# B&R Automation Studio project TD52 (part 91)

### Module_EngineGeneral.var - Module global variables
```iecst
VAR
	bAMM_2383 : BOOL := FALSE; (*ERROR: SAFETY - Exhaust gas backpressure high*) (*SAFETY PLC*) (*V04.14.00.00*)
	bAMM_2384 : BOOL := FALSE; (*ERROR: SAFETY - Speed deviation to ignition speed*) (*SAFETY PLC*) (*V04.14.00.00*)
	bAMM_2385 : BOOL := FALSE; (*ERROR: SAFETY - Ignition system failure*) (*SAFETY PLC*) (*V04.14.00.00*)
	bAMM_2386 : BOOL := FALSE; (*ERROR: SAFETY - Oil pressure minimum*) (*SAFETY PLC*) (*V04.14.00.00*)
	bAMM_2387 : BOOL := FALSE; (*ERROR: SAFETY - Oil pressure measuring signal failure*) (*SAFETY PLC*) (*V04.14.00.00*)
	bAMM_2388 : BOOL := FALSE; (*ERROR: SAFETY - Oil pressure implausible value*) (*SAFETY PLC*) (*V04.14.00.00*)
	bAMM_2389 : BOOL := FALSE; (*ERROR: SAFETY - Oil pressure deviation between the sensors*) (*SAFETY PLC*) (*V04.14.00.00*)
	bAMM_2390 : BOOL := FALSE; (*ERROR: SAFETY - Oil pressure maximum (sensor drift)*) (*SAFETY PLC*) (*V04.14.00.00*)
	bAMM_2391 : BOOL := FALSE; (*ERROR: SAFETY - Oil pressure sensor value frozen*) (*SAFETY PLC*) (*V04.14.00.00*)
	bAMM_2392 : BOOL := FALSE; (*ERROR: SAFETY - Oil pressure after pump maximum*) (*SAFETY PLC*) (*V04.14.00.00*)
	bAMM_2393 : BOOL := FALSE; (*ERROR: SAFETY - Oil pressure after pump measuring signal failure*) (*SAFETY PLC*) (*V04.14.00.00*)
	bAMM_2394 : BOOL := FALSE; (*ERROR: SAFETY - Oil pressure after pump implausible value*) (*SAFETY PLC*) (*V04.14.00.00*)
	bAMM_2395 : BOOL := FALSE; (*ERROR: SAFETY - Oil pressure after pump sensor value frozen*) (*SAFETY PLC*) (*V04.14.00.00*)
	bAMM_2396 : BOOL := FALSE; (*ERROR: SAFETY - Engine cooling water pressure minimum*) (*SAFETY PLC*) (*V04.14.00.00*)
	bAMM_2397 : BOOL := FALSE; (*ERROR: SAFETY - Engine cooling water pressure measuring signal failure*) (*SAFETY PLC*) (*V04.14.00.00*)
	bAMM_2398 : BOOL := FALSE; (*ERROR: SAFETY - Engine cooling water pressure deviation between the sensors*) (*SAFETY PLC*) (*V04.14.00.00*)
	bAMM_9408 : BOOL := FALSE; (*ERROR: SAFETY - Engine cooling water pressure maximum (sensor drift)*) (*SAFETY PLC*) (*V04.14.00.00*)
	bAMM_9409 : BOOL := FALSE; (*ERROR: SAFETY - Engine cooling water pressure sensor value frozen*) (*SAFETY PLC*) (*V04.14.00.00*)
	bAMM_9410 : BOOL := FALSE; (*ERROR: SAFETY - Engine cooling water pressure after pump maximum*) (*SAFETY PLC*) (*V04.14.00.00*)
	bAMM_9411 : BOOL := FALSE; (*ERROR: SAFETY - Engine cooling water pressure after pump measuring signal failure*) (*SAFETY PLC*) (*V04.14.00.00*)
	bAMM_9412 : BOOL := FALSE; (*ERROR: SAFETY - Engine cooling water pressure after pump sensor value frozen*) (*SAFETY PLC*) (*V04.14.00.00*)
	bAMM_9413 : BOOL := FALSE; (*ERROR: SAFETY - Generator circuit breaker opening failure*) (*SAFETY PLC*) (*V04.14.00.00*)
	bAMM_9414 : BOOL := FALSE; (*ERROR: SAFETY - Generator circuit breaker position feedback error*) (*SAFETY PLC*) (*V04.14.00.00*)
	bAMM_9415 : BOOL := FALSE; (*ERROR: SAFETY - Generator overload/short circuit*) (*SAFETY PLC*) (*V04.14.00.00*)
	bAMM_9416 : BOOL := FALSE; (*ERROR: SAFETY - Generator protection trip*) (*SAFETY PLC*) (*V04.14.00.00*)
	bAMM_9417 : BOOL := FALSE; (*ERROR: SAFETY - Collective fault in room ventilation*) (*SAFETY PLC*) (*V04.25.00.00*)
	bAMM_9418 : BOOL := FALSE; (*ERROR: SAFETY - Emergency stop push button - Module interface panel*) (*SAFETY PLC*) (*V04.14.00.00*)
	bAMM_9419 : BOOL := FALSE; (*ERROR: SAFETY - Emergency stop push button*) (*SAFETY PLC*) (*V04.14.00.00*)
	bAMM_9420 : BOOL := FALSE; (*ERROR: SAFETY - Safety loop 1 tripped - Module control panel*) (*SAFETY PLC*) (*V04.14.00.00*)
	bAMM_9421 : BOOL := FALSE; (*ERROR: SAFETY - Failure gas train 1*) (*SAFETY PLC*) (*V04.14.00.00*)
	bAMM_9422 : BOOL := FALSE; (*ERROR: SAFETY - Failure gas train 2*) (*SAFETY PLC*) (*V04.14.00.00*)
	bAMM_9423 : BOOL := FALSE; (*ERROR: SAFETY - Failure gas train 3*) (*SAFETY PLC*) (*V04.14.00.00*)
	bAMM_9424 : BOOL := FALSE; (*ERROR: SAFETY - Failure gas train 4*) (*SAFETY PLC*) (*V04.14.00.00*)
	bAMM_9425 : BOOL := FALSE; (*ERROR: SAFETY - Safety functions module interface panel - output not valid*) (*SAFETY PLC*) (*V04.14.00.00*)
	bAMM_9426 : BOOL := FALSE; (*ERROR: SAFETY - Safety functions module control panel - output not valid*) (*SAFETY PLC*) (*V04.14.00.00*)
	bAMM_9427 : BOOL := FALSE; (*ERROR: SAFETY - Engine type mismatch*) (*SAFETY PLC*) (*V04.14.00.00*)
	bAMM_9428 : BOOL := FALSE; (*ERROR: SAFETY - Room ventilation failure - Plausibility check pending*) (*SAFETY PLC*) (*V04.25.00.00*)
	bAMM_9429 : BOOL := FALSE; (*ERROR: SAFETY - Software handshake not valid*) (*SAFETY PLC*) (*V04.14.00.00*)
	bAMM_9430 : BOOL := FALSE; (*ERROR: SAFETY - Software not valid - Wrong CRC checksum*) (*SAFETY PLC*) (*V04.14.00.00*)
	bAMM_9431 : BOOL := FALSE; (*ERROR: SAFETY - Parameter mismatch*) (*SAFETY PLC*) (*V04.14.00.00*)
	bAMM_9433 : BOOL := FALSE; (*ERROR: SAFETY - Malfunction of safe communication channel *) (*SAFETY PLC*) (*V04.14.00.00*)
	bAMM_9434 : BOOL := FALSE; (*ERROR: SAFETY - Engine cooling water pump - Difference pressure minimum*) (*SAFETY PLC*) (*V04.25.00.00*)
	bAMM_9437 : BOOL := FALSE; (*ERROR: SAFETY - Scavenging flap not closed*) (*SAFETY PLC*) (*V04.25.00.00*)
	bAMM_9438 : BOOL := FALSE; (*ERROR: SAFETY - Scavenging flap failure*) (*SAFETY PLC*) (*V04.25.00.00*)
	bAMM_9439 : BOOL := FALSE; (*ERROR: SAFETY - Engine cooling water temperature after engine maximum*) (*SAFETY PLC*) (*V04.25.00.00*)
	bAMM_9440 : BOOL := FALSE; (*ERROR: SAFETY - Heating water supply temperature unit maximum*) (*SAFETY PLC*) (*V04.25.00.00*)
	bAMM_9441 : BOOL := FALSE; (*ERROR: SAFETY - Customer heating water circuit failure*) (*SAFETY PLC*) (*V04.25.00.00*)
	bAMM_9442 : BOOL := FALSE; (*ERROR: SAFETY - High temperature heating water level minimum*) (*SAFETY PLC*) (*V04.25.00.00*)
	bAMM_9443 : BOOL := FALSE; (*ERROR: SAFETY - High temperature heating water pressure 1 maximum*) (*SAFETY PLC*) (*V04.25.00.00*)
	bAMM_9444 : BOOL := FALSE; (*ERROR: SAFETY - High temperature heating water pressure 2 maximum*) (*SAFETY PLC*) (*V04.25.00.00*)
	bAMM_9445 : BOOL := FALSE; (*ERROR: SAFETY - High temperature heating water pressure 1 minimum*) (*SAFETY PLC*) (*V04.25.00.00*)
	bAMM_9446 : BOOL := FALSE; (*ERROR: SAFETY - High temperature heating water pressure 2 minimum*) (*SAFETY PLC*) (*V04.25.00.00*)
	bAMM_9447 : BOOL := FALSE; (*ERROR: SAFETY - High temperature heating water temperature 1 maximum*) (*SAFETY PLC*) (*V04.25.00.00*)
	bAMM_9448 : BOOL := FALSE; (*ERROR: SAFETY - High temperature heating water temperature 2 maximum*) (*SAFETY PLC*) (*V04.25.00.00*)
	bAMM_9449 : BOOL := FALSE; (*ERROR: SAFETY - High temperature heating water flow minimum*) (*SAFETY PLC*) (*V04.25.00.00*)
	bAMM_9450 : BOOL := FALSE; (*ERROR: SAFETY - Low temperature heating water level minimum*) (*SAFETY PLC*) (*V04.25.00.00*)
	bAMM_9451 : BOOL := FALSE; (*ERROR: SAFETY - Low temperature heating water pressure 1 maximum*) (*SAFETY PLC*) (*V04.25.00.00*)
	bAMM_9452 : BOOL := FALSE; (*ERROR: SAFETY - Low temperature heating water pressure 2 maximum*) (*SAFETY PLC*) (*V04.25.00.00*)
	bAMM_9453 : BOOL := FALSE; (*ERROR: SAFETY - Low temperature heating water pressure 1 minimum*) (*SAFETY PLC*) (*V04.25.00.00*)
	bAMM_9454 : BOOL := FALSE; (*ERROR: SAFETY - Low temperature heating water pressure 2 minimum*) (*SAFETY PLC*) (*V04.25.00.00*)
	bAMM_9455 : BOOL := FALSE; (*ERROR: SAFETY - Low temperature heating water temperature 1 maximum*) (*SAFETY PLC*) (*V04.25.00.00*)
	bAMM_9456 : BOOL := FALSE; (*ERROR: SAFETY - Low temperature heating water temperature 2 maximum*) (*SAFETY PLC*) (*V04.25.00.00*)
	bAMM_9457 : BOOL := FALSE; (*ERROR: SAFETY - Low temperature heating water flow minimum*) (*SAFETY PLC*) (*V04.25.00.00*)
	bAMM_9458 : BOOL := FALSE; (*ERROR: SAFETY - Safety loop 2 tripped - Module control panel*) (*SAFETY PLC*) (*V04.25.00.00*)
	bAMM_9459 : BOOL := FALSE; (*ERROR: SAFETY - Safety loop tripped - Module interface panel*) (*SAFETY PLC*) (*V04.25.00.00*)
	bAMM_9460 : BOOL := FALSE; (*ERROR: SAFETY - Emergency stop push button - Module control panel*) (*SAFETY PLC*) (*V04.25.00.00*)
	bAMM_9461 : BOOL := FALSE; (*ERROR: SAFETY - Emergency stop push button - Engine room button 1*) (*SAFETY PLC*) (*V04.25.00.00*)
	bAMM_9462 : BOOL := FALSE; (*ERROR: SAFETY - Emergency stop push button - Engine room button 2*) (*SAFETY PLC*) (*V04.25.00.00*)
	bAMM_9463 : BOOL := FALSE; (*ERROR: SAFETY - Emergency stop push button - Engine room button 3*) (*SAFETY PLC*) (*V04.25.00.00*)
	bAMM_9464 : BOOL := FALSE; (*ERROR: SAFETY - Emergency stop push button - Engine room button 4*) (*SAFETY PLC*) (*V04.25.00.00*)
	bAMM_9465 : BOOL := FALSE; (*ERROR: SAFETY - Emergency stop push button - External*) (*SAFETY PLC*) (*V04.25.00.00*)
	bAMM_9466 : BOOL := FALSE; (*ERROR: SAFETY - Emergency stop push button - Thermal reactor control panel*) (*SAFETY PLC*) (*V04.25.00.00*)
	bAMM_9467 : BOOL := FALSE; (*ERROR: SAFETY - Emergency stop push button - Interlock control panel*) (*SAFETY PLC*) (*V04.25.00.00*)
	bAMM_9468 : BOOL := FALSE; (*ERROR: SAFETY - Emergency stop push button - Master control panel*) (*SAFETY PLC*) (*V04.25.00.00*)
	bAMM_9469 : BOOL := FALSE; (*ERROR: SAFETY - Emergency stop push button - Exhaust gas after treatment control panel*) (*SAFETY PLC*) (*V04.25.00.00*)
	bAMM_9470 : BOOL := FALSE; (*ERROR: SAFETY - Emergency stop push button - Prechamber gas compressor*) (*SAFETY PLC*) (*V04.25.00.00*)
	bAMM_9471 : BOOL := FALSE; (*ERROR: SAFETY - Emergency stop push button - Auxiliaries control panel*) (*SAFETY PLC*) (*V04.25.00.00*)
	bAMM_9480 : BOOL := FALSE; (*ERROR: SAFETY - Room ventilation failure - Doors*) (*SAFETY PLC*) (*V04.25.00.00*)
	bAMM_9481 : BOOL := FALSE; (*ERROR: SAFETY - Room ventilation failure - Inlet air fan*) (*SAFETY PLC*) (*V04.25.00.00*)
	bAMM_9482 : BOOL := FALSE; (*ERROR: SAFETY - Room ventilation failure - Inlet air louvre*) (*SAFETY PLC*) (*V04.25.00.00*)
	bAMM_9483 : BOOL := FALSE; (*ERROR: SAFETY - Room ventilation failure - Outlet air louvre*) (*SAFETY PLC*) (*V04.25.00.00*)
	bAMM_9484 : BOOL := FALSE; (*ERROR: SAFETY - Failure gas train for decentral gas addition*) (*SAFETY PLC*) (*V04.25.00.00*)
	bAMM_9508 : BOOL := FALSE; (*WARNING: SAFETY - Malfunction of safe communication channel - Node 210*) (*SAFETY PLC*) (*V04.25.00.00*)
	bAMM_9514 : BOOL := FALSE; (*WARNING: SAFETY - Speed signal not valid*) (*SAFETY PLC*) (*V04.14.00.00*)
	bAMM_9515 : BOOL := FALSE; (*WARNING: SAFETY - Ignition plausibility check failure*) (*SAFETY PLC*) (*V04.14.00.00*)
	bAMM_9516 : BOOL := FALSE; (*WARNING: SAFETY - Ignition system running - signal not valid*) (*SAFETY PLC*) (*V04.14.00.00*)
	bAMM_9517 : BOOL := FALSE; (*WARNING: SAFETY - Release of synchronizing and load - output not valid*) (*SAFETY PLC*) (*V04.14.00.00*)
	bAMM_9518 : BOOL := FALSE; (*WARNING: SAFETY - Generator circuit breaker release undervoltage trip coil - output not valid*) (*SAFETY PLC*) (*V04.14.00.00*)
	bAMM_9519 : BOOL := FALSE; (*WARNING: SAFETY - Generator circuit breaker position ON - signal not valid*) (*SAFETY PLC*) (*V04.14.00.00*)
	bAMM_9520 : BOOL := FALSE; (*WARNING: SAFETY - Generator circuit breaker position OFF - signal not valid*) (*SAFETY PLC*) (*V04.14.00.00*)
	bAMM_9521 : BOOL := FALSE; (*WARNING: SAFETY - Generator overload/short circuit - signal not valid*) (*SAFETY PLC*) (*V04.14.00.00*)
	bAMM_9522 : BOOL := FALSE; (*WARNING: SAFETY - Generator protection trip - signal not valid*) (*SAFETY PLC*) (*V04.14.00.00*)
	bAMM_9523 : BOOL := FALSE; (*WARNING: SAFETY - Collective fault in room ventilation - plausibility check failure*) (*SAFETY PLC*) (*V04.25.00.00*)
	bAMM_9524 : BOOL := FALSE; (*WARNING: SAFETY - Collective fault in room ventilation - signal not valid*) (*SAFETY PLC*) (*V04.25.00.00*)
	bAMM_9525 : BOOL := FALSE; (*WARNING: SAFETY - Emergency stop push button - Module interface panel - signal not valid*) (*SAFETY PLC*) (*V04.14.00.00*)
	bAMM_9526 : BOOL := FALSE; (*WARNING: SAFETY - Emergency stop push button - signal not valid*) (*SAFETY PLC*) (*V04.14.00.00*)
	bAMM_9527 : BOOL := FALSE; (*WARNING: SAFETY - Safety loop 1 - Module control panel - signal not valid*) (*SAFETY PLC*) (*V04.14.00.00*)
	bAMM_9528 : BOOL := FALSE; (*WARNING: SAFETY - Release gas valve 1a - output not valid*) (*SAFETY PLC*) (*V04.14.00.00*)
	bAMM_9529 : BOOL := FALSE; (*WARNING: SAFETY - Release gas valve 1b - output not valid*) (*SAFETY PLC*) (*V04.14.00.00*)
	bAMM_9530 : BOOL := FALSE; (*WARNING: SAFETY - Release gas valve 2a - output not valid*) (*SAFETY PLC*) (*V04.14.00.00*)
	bAMM_9531 : BOOL := FALSE; (*WARNING: SAFETY - Release gas valve 2b - output not valid*) (*SAFETY PLC*) (*V04.14.00.00*)
	bAMM_9532 : BOOL := FALSE; (*WARNING: SAFETY - Release gas valve 3a - output not valid*) (*SAFETY PLC*) (*V04.14.00.00*)
	bAMM_9533 : BOOL := FALSE; (*WARNING: SAFETY - Release gas valve 3b - output not valid*) (*SAFETY PLC*) (*V04.14.00.00*)
	bAMM_9534 : BOOL := FALSE; (*WARNING: SAFETY - Release gas valve 4a - output not valid*) (*SAFETY PLC*) (*V04.14.00.00*)
	bAMM_9535 : BOOL := FALSE; (*WARNING: SAFETY - Release gas valve 4b - output not valid*) (*SAFETY PLC*) (*V04.14.00.00*)
	bAMM_9536 : BOOL := FALSE; (*WARNING: SAFETY - Gas safety device 1 - signal not valid*) (*SAFETY PLC*) (*V04.14.00.00*)
	bAMM_9537 : BOOL := FALSE; (*WARNING: SAFETY - Gas safety device 2 - signal not valid*) (*SAFETY PLC*) (*V04.14.00.00*)
	bAMM_9538 : BOOL := FALSE; (*WARNING: SAFETY - Gas safety device 3 - signal not valid*) (*SAFETY PLC*) (*V04.14.00.00*)
	bAMM_9539 : BOOL := FALSE; (*WARNING: SAFETY - Gas safety device 4 - signal not valid*) (*SAFETY PLC*) (*V04.14.00.00*)
	bAMM_9540 : BOOL := FALSE; (*WARNING: SAFETY - Gas safety device 1 - output not valid*) (*SAFETY PLC*) (*V04.14.00.00*)
	bAMM_9541 : BOOL := FALSE; (*WARNING: SAFETY - Gas safety device 2 - output not valid*) (*SAFETY PLC*) (*V04.14.00.00*)
	bAMM_9542 : BOOL := FALSE; (*WARNING: SAFETY - Gas safety device 3 - output not valid*) (*SAFETY PLC*) (*V04.14.00.00*)
	bAMM_9543 : BOOL := FALSE; (*WARNING: SAFETY - Gas safety device 4 - output not valid*) (*SAFETY PLC*) (*V04.14.00.00*)
	bAMM_9544 : BOOL := FALSE; (*WARNING: SAFETY - Malfunction of safe communication channel - Node 101*) (*SAFETY PLC*) (*V04.14.00.00*)
	bAMM_9545 : BOOL := FALSE; (*WARNING: SAFETY - Malfunction of safe communication channel - Node 102*) (*SAFETY PLC*) (*V04.14.00.00*)
	bAMM_9546 : BOOL := FALSE; (*WARNING: SAFETY - Malfunction of safe communication channel - Node 103*) (*SAFETY PLC*) (*V04.14.00.00*)
	bAMM_9547 : BOOL := FALSE; (*WARNING: SAFETY - Malfunction of safe communication channel - Node 104*) (*SAFETY PLC*) (*V04.14.00.00*)
	bAMM_9548 : BOOL := FALSE; (*WARNING: SAFETY - Malfunction of safe communication channel - Node 201*) (*SAFETY PLC*) (*V04.14.00.00*)
	bAMM_9549 : BOOL := FALSE; (*WARNING: SAFETY - Malfunction of safe communication channel - Node 202*) (*SAFETY PLC*) (*V04.14.00.00*)
	bAMM_9550 : BOOL := FALSE; (*WARNING: SAFETY - Malfunction of safe communication channel - Node 203*) (*SAFETY PLC*) (*V04.14.00.00*)
	bAMM_9551 : BOOL := FALSE; (*WARNING: SAFETY - Malfunction of safe communication channel - Node 204*) (*SAFETY PLC*) (*V04.14.00.00*)
	bAMM_9552 : BOOL := FALSE; (*WARNING: SAFETY - Malfunction of safe communication channel - Node 205*) (*SAFETY PLC*) (*V04.14.00.00*)
	bAMM_9553 : BOOL := FALSE; (*WARNING: SAFETY - Malfunction of safe communication channel - Node 206*) (*SAFETY PLC*) (*V04.14.00.00*)
	bAMM_9554 : BOOL := FALSE; (*WARNING: SAFETY - Malfunction of safe communication channel - Node 207*) (*SAFETY PLC*) (*V04.14.00.00*)
	bAMM_9555 : BOOL := FALSE; (*WARNING: SAFETY - Malfunction of safe communication channel - Node 208*) (*SAFETY PLC*) (*V04.14.00.00*)
	bAMM_9556 : BOOL := FALSE; (*WARNING: SAFETY - Malfunction of safe communication channel - Node 209*) (*SAFETY PLC*) (*V04.14.00.00*)
	bAMM_9562 : BOOL := FALSE; (*WARNING: SAFETY - Scavenging flap plausibility check failure*) (*SAFETY PLC*) (*V04.25.00.00*)
	bAMM_9563 : BOOL := FALSE; (*WARNING: SAFETY - Scavenging flap closed feedback - signal not valid*) (*SAFETY PLC*) (*V04.25.00.00*)
	bAMM_9564 : BOOL := FALSE; (*WARNING: SAFETY - Scavenging flap temperature switch - signal not valid*) (*SAFETY PLC*) (*V04.25.00.00*)
	bAMM_9565 : BOOL := FALSE; (*WARNING: SAFETY - Customer heating water circuit failure - signal not valid*) (*SAFETY PLC*) (*V04.25.00.00*)
	bAMM_9566 : BOOL := FALSE; (*WARNING: SAFETY - High temperature heating water flow minimum - plausibility check failure*) (*SAFETY PLC*) (*V04.25.00.00*)
	bAMM_9567 : BOOL := FALSE; (*WARNING: SAFETY - High temperature heating water level minimum - signal not valid*) (*SAFETY PLC*) (*V04.25.00.00*)
	bAMM_9568 : BOOL := FALSE; (*WARNING: SAFETY - High temperature heating water pressure 1 maximum - signal not valid*) (*SAFETY PLC*) (*V04.25.00.00*)
	bAMM_9569 : BOOL := FALSE; (*WARNING: SAFETY - High temperature heating water pressure 2 maximum - signal not valid*) (*SAFETY PLC*) (*V04.25.00.00*)
	bAMM_9570 : BOOL := FALSE; (*WARNING: SAFETY - High temperature heating water pressure 1 minimum - signal not valid*) (*SAFETY PLC*) (*V04.25.00.00*)
	bAMM_9571 : BOOL := FALSE; (*WARNING: SAFETY - High temperature heating water pressure 2 minimum - signal not valid*) (*SAFETY PLC*) (*V04.25.00.00*)
	bAMM_9572 : BOOL := FALSE; (*WARNING: SAFETY - High temperature heating water temperature 1 maximum - signal not valid*) (*SAFETY PLC*) (*V04.25.00.00*)
	bAMM_9573 : BOOL := FALSE; (*WARNING: SAFETY - High temperature heating water temperature 2 maximum - signal not valid*) (*SAFETY PLC*) (*V04.25.00.00*)
	bAMM_9574 : BOOL := FALSE; (*WARNING: SAFETY - High temperature heating water flow minimum - signal not valid*) (*SAFETY PLC*) (*V04.25.00.00*)
	bAMM_9575 : BOOL := FALSE; (*WARNING: SAFETY - Low temperature heating water flow minimum - plausibility check failure*) (*SAFETY PLC*) (*V04.25.00.00*)
	bAMM_9576 : BOOL := FALSE; (*WARNING: SAFETY - Low temperature heating water level minimum - signal not valid*) (*SAFETY PLC*) (*V04.25.00.00*)
	bAMM_9577 : BOOL := FALSE; (*WARNING: SAFETY - Low temperature heating water pressure 1 maximum - signal not valid*) (*SAFETY PLC*) (*V04.25.00.00*)
	bAMM_9578 : BOOL := FALSE; (*WARNING: SAFETY - Low temperature heating water pressure 2 maximum - signal not valid*) (*SAFETY PLC*) (*V04.25.00.00*)
	bAMM_9579 : BOOL := FALSE; (*WARNING: SAFETY - Low temperature heating water pressure 1 minimum - signal not valid*) (*SAFETY PLC*) (*V04.25.00.00*)
	bAMM_9580 : BOOL := FALSE; (*WARNING: SAFETY - Low temperature heating water pressure 2 minimum - signal not valid*) (*SAFETY PLC*) (*V04.25.00.00*)
	bAMM_9581 : BOOL := FALSE; (*WARNING: SAFETY - Low temperature heating water temperature 1 maximum - signal not valid*) (*SAFETY PLC*) (*V04.25.00.00*)
	bAMM_9582 : BOOL := FALSE; (*WARNING: SAFETY - Low temperature heating water temperature 2 maximum - signal not valid*) (*SAFETY PLC*) (*V04.25.00.00*)
	bAMM_9583 : BOOL := FALSE; (*WARNING: SAFETY - Low temperature heating water flow minimum - signal not valid*) (*SAFETY PLC*) (*V04.25.00.00*)
	bAMM_9584 : BOOL := FALSE; (*WARNING: SAFETY - Safety loop 2 - Module control panel - signal not valid*) (*SAFETY PLC*) (*V04.25.00.00*)
	bAMM_9585 : BOOL := FALSE; (*WARNING: SAFETY - Safety loop - Module interface panel - signal not valid*) (*SAFETY PLC*) (*V04.25.00.00*)
	bAMM_9586 : BOOL := FALSE; (*WARNING: SAFETY - Exhaust gas backpressure high - signal not valid*) (*SAFETY PLC*) (*V04.25.00.00*)
	bAMM_9587 : BOOL := FALSE; (*WARNING: SAFETY - Emergency stop signalling - output not valid*) (*SAFETY PLC*) (*V04.25.00.00*)
	bAMM_9593 : BOOL := FALSE; (*WARNING: SAFETY - Nominal speed mismatch*) (*SAFETY PLC*) (*V04.25.00.00*)
	bAMM_9597 : BOOL := FALSE; (*WARNING: SAFETY - Malfunction of safe communication channel - Node 300*) (*SAFETY PLC*) (*V04.25.00.00*)
	bAMM_9598 : BOOL := FALSE; (*WARNING: SAFETY - Malfunction of safe communication channel - Node 301*) (*SAFETY PLC*) (*V04.25.00.00*)
	bAMM_9600 : BOOL := FALSE; (*WARNING: SAFETY - Malfunction of safe communication channel - Node 105*) (*SAFETY PLC*) (*V04.25.00.00*)
	bAMM_9627 : BOOL := FALSE; (*WARNING: SAFETY - Room ventilation failure - Doors - plausibility check failure*) (*SAFETY PLC*) (*V04.25.00.00*)
	bAMM_9628 : BOOL := FALSE; (*WARNING: SAFETY - Room ventilation failure - Doors - signal not valid*) (*SAFETY PLC*) (*V04.25.00.00*)
	bAMM_9629 : BOOL := FALSE; (*WARNING: SAFETY - Room ventilation failure - Inlet air fan group 1*) (*SAFETY PLC*) (*V04.25.00.00*)
	bAMM_9630 : BOOL := FALSE; (*WARNING: SAFETY - Room ventilation failure - Inlet air fan group 1 - plausibility check failure*) (*SAFETY PLC*) (*V04.25.00.00*)
	bAMM_9631 : BOOL := FALSE; (*WARNING: SAFETY - Room ventilation failure - Inlet air fan group 1 - signal not valid*) (*SAFETY PLC*) (*V04.25.00.00*)
	bAMM_9632 : BOOL := FALSE; (*WARNING: SAFETY - Room ventilation failure - Inlet air fan group 2*) (*SAFETY PLC*) (*V04.25.00.00*)
	bAMM_9633 : BOOL := FALSE; (*WARNING: SAFETY - Room ventilation failure - Inlet air fan group 2 - plausibility check failure*) (*SAFETY PLC*) (*V04.25.00.00*)
	bAMM_9634 : BOOL := FALSE; (*WARNING: SAFETY - Room ventilation failure - Inlet air fan group 2 - signal not valid*) (*SAFETY PLC*) (*V04.25.00.00*)
	bAMM_9635 : BOOL := FALSE; (*WARNING: SAFETY - Room ventilation failure - Inlet air fan group 3*) (*SAFETY PLC*) (*V04.25.00.00*)
	bAMM_9636 : BOOL := FALSE; (*WARNING: SAFETY - Room ventilation failure - Inlet air fan group 3 - plausibility check failure*) (*SAFETY PLC*) (*V04.25.00.00*)
	bAMM_9637 : BOOL := FALSE; (*WARNING: SAFETY - Room ventilation failure - Inlet air fan group 3 - signal not valid*) (*SAFETY PLC*) (*V04.25.00.00*)
	bAMM_9638 : BOOL := FALSE; (*WARNING: SAFETY - Room ventilation failure - Inlet air fan group 4*) (*SAFETY PLC*) (*V04.25.00.00*)
	bAMM_9639 : BOOL := FALSE; (*WARNING: SAFETY - Room ventilation failure - Inlet air fan group 4 - plausibility check failure*) (*SAFETY PLC*) (*V04.25.00.00*)
	bAMM_9640 : BOOL := FALSE; (*WARNING: SAFETY - Room ventilation failure - Inlet air fan group 4 - signal not valid*) (*SAFETY PLC*) (*V04.25.00.00*)
	bAMM_9641 : BOOL := FALSE; (*WARNING: SAFETY - Room ventilation failure - Inlet air fan group 5*) (*SAFETY PLC*) (*V04.25.00.00*)
	bAMM_9642 : BOOL := FALSE; (*WARNING: SAFETY - Room ventilation failure - Inlet air fan group 5 - plausibility check failure*) (*SAFETY PLC*) (*V04.25.00.00*)
	bAMM_9643 : BOOL := FALSE; (*WARNING: SAFETY - Room ventilation failure - Inlet air fan group 5 - signal not valid*) (*SAFETY PLC*) (*V04.25.00.00*)
	bAMM_9644 : BOOL := FALSE; (*WARNING: SAFETY - Room ventilation failure - Inlet air fan group 6*) (*SAFETY PLC*) (*V04.25.00.00*)
	bAMM_9645 : BOOL := FALSE; (*WARNING: SAFETY - Room ventilation failure - Inlet air fan group 6 - plausibility check failure*) (*SAFETY PLC*) (*V04.25.00.00*)
	bAMM_9646 : BOOL := FALSE; (*WARNING: SAFETY - Room ventilation failure - Inlet air fan group 6 - signal not valid*) (*SAFETY PLC*) (*V04.25.00.00*)
	bAMM_9647 : BOOL := FALSE; (*WARNING: SAFETY - Room ventilation failure - Inlet air louvre group 1 - opened signal*) (*SAFETY PLC*) (*V04.25.00.00*)
	bAMM_9648 : BOOL := FALSE; (*WARNING: SAFETY - Room ventilation failure - Inlet air louvre group 1 - closed signal*) (*SAFETY PLC*) (*V04.25.00.00*)
	bAMM_9649 : BOOL := FALSE; (*WARNING: SAFETY - Room ventilation failure - Inlet air louvre group 1 - opened signal not valid*) (*SAFETY PLC*) (*V04.25.00.00*)
	bAMM_9650 : BOOL := FALSE; (*WARNING: SAFETY - Room ventilation failure - Inlet air louvre group 1 - closed signal not valid*) (*SAFETY PLC*) (*V04.25.00.00*)
	bAMM_9651 : BOOL := FALSE; (*WARNING: SAFETY - Room ventilation failure - Inlet air louvre group 1 - plausibility check failure*) (*SAFETY PLC*) (*V04.25.00.00*)
	bAMM_9652 : BOOL := FALSE; (*WARNING: SAFETY - Room ventilation failure - Inlet air louvre group 2 - opened signal*) (*SAFETY PLC*) (*V04.25.00.00*)
	bAMM_9653 : BOOL := FALSE; (*WARNING: SAFETY - Room ventilation failure - Inlet air louvre group 2 - closed signal*) (*SAFETY PLC*) (*V04.25.00.00*)
	bAMM_9654 : BOOL := FALSE; (*WARNING: SAFETY - Room ventilation failure - Inlet air louvre group 2 - opened signal not valid*) (*SAFETY PLC*) (*V04.25.00.00*)
	bAMM_9655 : BOOL := FALSE; (*WARNING: SAFETY - Room ventilation failure - Inlet air louvre group 2 - closed signal not valid*) (*SAFETY PLC*) (*V04.25.00.00*)
	bAMM_9656 : BOOL := FALSE; (*WARNING: SAFETY - Room ventilation failure - Inlet air louvre group 2 - plausibility check failure*) (*SAFETY PLC*) (*V04.25.00.00*)
	bAMM_9657 : BOOL := FALSE; (*WARNING: SAFETY - Room ventilation failure - Inlet air louvre group 3 - opened signal*) (*SAFETY PLC*) (*V04.25.00.00*)
	bAMM_9658 : BOOL := FALSE; (*WARNING: SAFETY - Room ventilation failure - Inlet air louvre group 3 - closed signal*) (*SAFETY PLC*) (*V04.25.00.00*)
	bAMM_9659 : BOOL := FALSE; (*WARNING: SAFETY - Room ventilation failure - Inlet air louvre group 3 - opened signal not valid*) (*SAFETY PLC*) (*V04.25.00.00*)
	bAMM_9660 : BOOL := FALSE; (*WARNING: SAFETY - Room ventilation failure - Inlet air louvre group 3 - closed signal not valid*) (*SAFETY PLC*) (*V04.25.00.00*)
	bAMM_9661 : BOOL := FALSE; (*WARNING: SAFETY - Room ventilation failure - Inlet air louvre group 3 - plausibility check failure*) (*SAFETY PLC*) (*V04.25.00.00*)
	bAMM_9662 : BOOL := FALSE; (*WARNING: SAFETY - Room ventilation failure - Inlet air louvre group 4 - opened signal*) (*SAFETY PLC*) (*V04.25.00.00*)
	bAMM_9663 : BOOL := FALSE; (*WARNING: SAFETY - Room ventilation failure - Inlet air louvre group 4 - closed signal*) (*SAFETY PLC*) (*V04.25.00.00*)
	bAMM_9664 : BOOL := FALSE; (*WARNING: SAFETY - Room ventilation failure - Inlet air louvre group 4 - opened signal not valid*) (*SAFETY PLC*) (*V04.25.00.00*)
	bAMM_9665 : BOOL := FALSE; (*WARNING: SAFETY - Room ventilation failure - Inlet air louvre group 4 - closed signal not valid*) (*SAFETY PLC*) (*V04.25.00.00*)
	bAMM_9666 : BOOL := FALSE; (*WARNING: SAFETY - Room ventilation failure - Inlet air louvre group 4 - plausibility check failure*) (*SAFETY PLC*) (*V04.25.00.00*)
	bAMM_9667 : BOOL := FALSE; (*WARNING: SAFETY - Room ventilation failure - Inlet air louvre group 5 - opened signal*) (*SAFETY PLC*) (*V04.25.00.00*)
	bAMM_9668 : BOOL := FALSE; (*WARNING: SAFETY - Room ventilation failure - Inlet air louvre group 5 - closed signal*) (*SAFETY PLC*) (*V04.25.00.00*)
	bAMM_9669 : BOOL := FALSE; (*WARNING: SAFETY - Room ventilation failure - Inlet air louvre group 5 - opened signal not valid*) (*SAFETY PLC*) (*V04.25.00.00*)
	bAMM_9670 : BOOL := FALSE; (*WARNING: SAFETY - Room ventilation failure - Inlet air louvre group 5 - closed signal not valid*) (*SAFETY PLC*) (*V04.25.00.00*)
	bAMM_9671 : BOOL := FALSE; (*WARNING: SAFETY - Room ventilation failure - Inlet air louvre group 5 - plausibility check failure*) (*SAFETY PLC*) (*V04.25.00.00*)
	bAMM_9672 : BOOL := FALSE; (*WARNING: SAFETY - Room ventilation failure - Inlet air louvre group 6 - opened signal*) (*SAFETY PLC*) (*V04.25.00.00*)
	bAMM_9673 : BOOL := FALSE; (*WARNING: SAFETY - Room ventilation failure - Inlet air louvre group 6 - closed signal*) (*SAFETY PLC*) (*V04.25.00.00*)
	bAMM_9674 : BOOL := FALSE; (*WARNING: SAFETY - Room ventilation failure - Inlet air louvre group 6 - opened signal not valid*) (*SAFETY PLC*) (*V04.25.00.00*)
	bAMM_9675 : BOOL := FALSE; (*WARNING: SAFETY - Room ventilation failure - Inlet air louvre group 6 - closed signal not valid*) (*SAFETY PLC*) (*V04.25.00.00*)
	bAMM_9676 : BOOL := FALSE; (*WARNING: SAFETY - Room ventilation failure - Inlet air louvre group 6 - plausibility check failure*) (*SAFETY PLC*) (*V04.25.00.00*)
	bAMM_9677 : BOOL := FALSE; (*WARNING: SAFETY - Room ventilation failure - Outlet air louvre group 1 - closed signal*) (*SAFETY PLC*) (*V04.25.00.00*)
	bAMM_9678 : BOOL := FALSE; (*WARNING: SAFETY - Room ventilation failure - Outlet air louvre group 1 - opened signal not valid*) (*SAFETY PLC*) (*V04.25.00.00*)
	bAMM_9679 : BOOL := FALSE; (*WARNING: SAFETY - Room ventilation failure - Outlet air louvre group 1 - closed signal not valid*) (*SAFETY PLC*) (*V04.25.00.00*)
	bAMM_9680 : BOOL := FALSE; (*WARNING: SAFETY - Room ventilation failure - Outlet air louvre group 1 - plausibility check failure*) (*SAFETY PLC*) (*V04.25.00.00*)
	bAMM_9681 : BOOL := FALSE; (*WARNING: SAFETY - Room ventilation failure - Outlet air louvre group 2 - closed signal*) (*SAFETY PLC*) (*V04.25.00.00*)
	bAMM_9682 : BOOL := FALSE; (*WARNING: SAFETY - Room ventilation failure - Outlet air louvre group 2 - opened signal not valid*) (*SAFETY PLC*) (*V04.25.00.00*)
	bAMM_9683 : BOOL := FALSE; (*WARNING: SAFETY - Room ventilation failure - Outlet air louvre group 2 - closed signal not valid*) (*SAFETY PLC*) (*V04.25.00.00*)
	bAMM_9684 : BOOL := FALSE; (*WARNING: SAFETY - Room ventilation failure - Outlet air louvre group 2 - plausibility check failure*) (*SAFETY PLC*) (*V04.25.00.00*)
	bAMM_9685 : BOOL := FALSE; (*WARNING: SAFETY - Room ventilation failure - Outlet air louvre group 3 - closed signal*) (*SAFETY PLC*) (*V04.25.00.00*)
	bAMM_9686 : BOOL := FALSE; (*WARNING: SAFETY - Room ventilation failure - Outlet air louvre group 3 - opened signal not valid*) (*SAFETY PLC*) (*V04.25.00.00*)
	bAMM_9687 : BOOL := FALSE; (*WARNING: SAFETY - Room ventilation failure - Outlet air louvre group 3 - closed signal not valid*) (*SAFETY PLC*) (*V04.25.00.00*)
	bAMM_9688 : BOOL := FALSE; (*WARNING: SAFETY - Room ventilation failure - Outlet air louvre group 3 - plausibility check failure*) (*SAFETY PLC*) (*V04.25.00.00*)
	bAMM_9689 : BOOL := FALSE; (*WARNING: SAFETY - Room ventilation failure - Outlet air louvre group 4 - closed signal*) (*SAFETY PLC*) (*V04.25.00.00*)
	bAMM_9690 : BOOL := FALSE; (*WARNING: SAFETY - Room ventilation failure - Outlet air louvre group 4 - opened signal not valid*) (*SAFETY PLC*) (*V04.25.00.00*)
	bAMM_9691 : BOOL := FALSE; (*WARNING: SAFETY - Room ventilation failure - Outlet air louvre group 4 - closed signal not valid*) (*SAFETY PLC*) (*V04.25.00.00*)
	bAMM_9692 : BOOL := FALSE; (*WARNING: SAFETY - Room ventilation failure - Outlet air louvre group 4 - plausibility check failure*) (*SAFETY PLC*) (*V04.25.00.00*)
	bAMM_9693 : BOOL := FALSE; (*WARNING: SAFETY - Room ventilation failure - Outlet air louvre group 5 - closed signal*) (*SAFETY PLC*) (*V04.25.00.00*)
	bAMM_9694 : BOOL := FALSE; (*WARNING: SAFETY - Room ventilation failure - Outlet air louvre group 5 - opened signal not valid*) (*SAFETY PLC*) (*V04.25.00.00*)
	bAMM_9695 : BOOL := FALSE; (*WARNING: SAFETY - Room ventilation failure - Outlet air louvre group 5 - closed signal not valid*) (*SAFETY PLC*) (*V04.25.00.00*)
	bAMM_9696 : BOOL := FALSE; (*WARNING: SAFETY - Room ventilation failure - Outlet air louvre group 5 - plausibility check failure*) (*SAFETY PLC*) (*V04.25.00.00*)
	bAMM_9697 : BOOL := FALSE; (*WARNING: SAFETY - Room ventilation failure - Outlet air louvre group 6 - closed signal*) (*SAFETY PLC*) (*V04.25.00.00*)
	bAMM_9698 : BOOL := FALSE; (*WARNING: SAFETY - Room ventilation failure - Outlet air louvre group 6 - opened signal not valid*) (*SAFETY PLC*) (*V04.25.00.00*)
	bAMM_9699 : BOOL := FALSE; (*WARNING: SAFETY - Room ventilation failure - Outlet air louvre group 6 - closed signal not valid*) (*SAFETY PLC*) (*V04.25.00.00*)
	bAMM_9700 : BOOL := FALSE; (*WARNING: SAFETY - Room ventilation failure - Outlet air louvre group 6 - plausibility check failure*) (*SAFETY PLC*) (*V04.25.00.00*)
	bAMM_9701 : BOOL := FALSE; (*WARNING: SAFETY - Release gas valve A for decentral gas addition - output not valid*) (*SAFETY PLC*) (*V04.25.00.00*)
	bAMM_9702 : BOOL := FALSE; (*WARNING: SAFETY - Release gas valve B for decentral gas addition - output not valid*) (*SAFETY PLC*) (*V04.25.00.00*)
	bAMM_9703 : BOOL := FALSE; (*WARNING: SAFETY - Gas safety device for decentral gas addition - signal not valid*) (*SAFETY PLC*) (*V04.25.00.00*)
	bAMM_9704 : BOOL := FALSE; (*WARNING: SAFETY - Gas safety device for decentral gas addition - output not valid*) (*SAFETY PLC*) (*V04.25.00.00*)
	bAMM_IdleFriction_HiHi : BOOL := FALSE; (*idle friction to high - error*) (* *) (*V04.04.00.00*)
	bAMM_Pr_Baro_Ms : BOOL := FALSE; (*barometric pressure - measurement signal failure*) (* *) (*V04.02.00.00*)
	bAMM_Pr_Baro_siteDev_Hi : BOOL := FALSE; (*barometric pressure maximum - warning*) (* *) (*V04.02.00.00*)
	bAMM_Pr_Baro_siteDev_Lo : BOOL := FALSE; (*barometric pressure minimum - warning*) (* *) (*V04.02.00.00*)
	bAMM_PUscuff : BOOL := FALSE; (*PU scuffing detection - alarm*) (* *) (*V04.11.00.00*)
	bAMM_SlowDownTime_LoLo : BOOL := FALSE; (*ERROR slow down time too short*) (* *) (*V04.01.00.00*)
	bAMM_SlowDownTime_LoLo_Save : BOOL := FALSE; (*ERROR slow down time too short -  restore after cold start of CPU*) (* *) (*V04.07.00.00*)
	bAMM_T_CBearing_Calib : BOOL := FALSE; (*conrod bearing temperature calibration unsuccessful - warning*) (* *) (*V04.04.00.00*)
	bAMM_T_CBearing_CAN : BOOL := FALSE; (*conrod bearing temperature CAN bus communication - error*) (* *) (*V04.02.00.00*)
	bAMM_T_CBearing_Hi : BOOL := FALSE; (*conrod bearing temperature maximum - warning*) (* *) (*V04.02.00.00*)
	bAMM_T_CBearing_HiHi : BOOL := FALSE; (*conrod bearing temperature maximum - error*) (* *) (*V04.02.00.00*)
	bAMM_T_CBearing_MDev_HiHi : BOOL := FALSE; (*conrod bearing temperature - positive deviation from MEDIAN maximum - error*) (* *) (*V04.02.00.00*)
	bAMM_T_CBearing_MDev_Lo : BOOL := FALSE; (*conrod bearing temperature - negative deviation from MEDIAN maximum - error*) (* *) (*V04.05.01.00*)
	bAMM_T_CBearing_Ms : BOOL := FALSE; (*conrod bearing temperature measuring signal failure*) (* *) (*V04.04.00.00*)
	bAMM_T_CBearing_Sig_Lo : BOOL := FALSE; (*conrod bearing signal intensity minimum - warning*) (* *) (*V04.04.00.00*)
	bAMM_T_MBearing_Hi : BOOL := FALSE; (*main bearing temperature maximum - warning*) (* *) (*V04.02.00.00*)
	bAMM_T_MBearing_HiHi : BOOL := FALSE; (*main bearing temperature maximum - error*) (* *) (*V04.02.00.00*)
	bAMM_T_MBearing_MDev_HiHi : BOOL := FALSE; (*main bearing temperature - positive deviation from MEDIAN maximum - error*) (* *) (*V04.02.00.00*)
	bAMM_T_MBearing_MDev_Lo : BOOL := FALSE; (*main bearing temperature - negative deviation from MEDIAN maximum - warning*) (* *) (*V04.05.01.00*)
	bAMM_T_MBearing_Ms : BOOL := FALSE; (*main bearing temperature measuring signal failure - warning*) (* *) (*V04.05.01.00*)
	bErrPermSlowDown : BOOL := FALSE; (*ERROR permanent memory Slowdown time*) (* *) (*V04.01.00.00*)
	bGnlTrip : BOOL; (*general alarm trip *)
	bGnlTrip1 : BOOL; (*general alarm trip priority 1*)
	bGnlTrip2 : BOOL; (*general alarm trip priority 2*)
	bGnlTrip3 : BOOL; (*general alarm trip priority 3*)
	bGnlWarning : BOOL; (*general alarm warning *)
	bMsg2285_Test : BOOL := FALSE; (*alarm bypass of A2285 main bearing temperature - positive deviation from average value*) (* *) (*V04.05.03.00*)
	bMsg2286_Test : BOOL := FALSE; (*alarm bypass of A2286 conrod bearing temperature - positive deviation from average value*) (* *) (*V04.05.03.00*)
	bNoInitDetected : BOOL := FALSE; (*allways true, except 1cycle on init up*)
	bOMSS_MAT : BOOL; (*operation mode selector switch - MANUAL/AUTO/TEST*) (* *) (*V04.02.00.00*)
	bOpM_PUscuff : BOOL := FALSE; (*PU scuffing detection - operating message*) (* *) (*V04.11.00.00*)
	bOpM_T_CBearing_Calib_Ok : BOOL := FALSE; (*conrod bearing temperature calibration successful - operating message*) (* *) (*V04.05.00.00*)
	bOpM_T_CBearing_Hi : BOOL := FALSE; (*conrod bearing temperature maximum - operating message*) (* *) (*V04.02.00.00*)
	bOpM_T_CBearing_MDev_HiHi : BOOL := FALSE; (*conrod bearing temperature - positive deviation from MEDIAN maximum - operating message*) (* *) (*V04.04.00.00*)
	bOpM_T_CBearing_MDev_Lo : BOOL := FALSE; (*conrod bearing temperature - negative deviation from MEDIAN maximum - operating message*) (* *) (*V04.05.01.00*)
	bOpM_T_CBearing_Ms : BOOL := FALSE; (*conrod bearing temperature measuring signal failure - operating message*) (* *) (*V04.02.00.00*)
	bOpM_T_CBearing_Sig_Lo : BOOL := FALSE; (*conrod bearing signal intensity minimum - operating message*) (* *) (*V04.04.00.00*)
	bOpM_T_MBearing_Hi : BOOL := FALSE; (*main bearing temperature maximum - operating message*) (* *) (*V04.02.00.00*)
	bOpM_T_MBearing_MDev_HiHi : BOOL := FALSE; (*main bearing temperature - positive deviation from MEDIAN maximum - operating message*) (* *) (*V04.04.00.00*)
	bOpM_T_MBearing_MDev_Lo : BOOL := FALSE; (*main bearing temperature - negative deviation from MEDIAN maximum - operating message*) (* *) (*V04.05.01.00*)
	bOpM_T_MBearing_Ms : BOOL := FALSE; (*main bearing temperature measuring signal failure - operating message*) (* *) (*V04.05.01.00*)
	bP_Lo_Trig : BOOL := FALSE; (*Power signal missing ( lower 10%)*)
	bRelModul_ParaSetupOk : BOOL := FALSE; (*Release Module if ParaSetupOk = TRUE*) (* *) (*V04.03.00.00*)
	bStartSpd : BOOL := FALSE; (*actual engine speed > start speed*)
	IN_EG : IN_EG_Struct; (*Module IN-Interface*)
	MM2VIS : MM2VIS_Struct; (*Module VISU-Interface (Module --> VISU)*)
	OUT_EG : OUT_EG_Struct; (*Module OUT-Interface*)
	Para : PARA_EG_Struct; (*Module Parameter-Interface*)
	ParaFactoryDefault : PARA_EG_Struct := (0); (*First Init Values*)
	pm : PARA_EG_Struct; (*Stored parameter structure *)
	VIS2MM : VIS2MM_Struct; (*Module VISU-Interface (VISU --> Module)*)
	xEngType : EngType; (*Instance of FB EngType*)
	xOpMode : OpMode; (*Function block for operation mode*) (* *) (*V04.10.00.00*)
	xPUscuff : fPUscuff; (*Function block for PU scuffing detection*) (* *) (*V04.11.00.00*)
END_VAR
```

### sPLC.typ - SAFETY PLC data types
```iecst
TYPE
	MM2VIS_sPLC_Struct : 	STRUCT
		bCompletion_Busy : BOOL;
		bCompletion_Done : BOOL;
		bCompletion_Error : BOOL;
		bConnect_Active : BOOL;
		bConnect_Busy : BOOL;
		bConnect_Error : BOOL;
		bControl_Busy : BOOL;
		bControl_Done : BOOL;
		bControl_Error : BOOL;
		bExchange_Busy : BOOL;
		bExchange_Done : BOOL;
		bExchange_Error : BOOL;
		bF02_DI_Ign_Run : BOOL; (*Function 02 - Digital Input - Feedback Ignition*)
		bF07_DI_GCB_Off : BOOL; (*Function 07 - Digital Input - Generator circuit breaker opened*)
		bF07_DI_GCB_On : BOOL; (*Function 07 - Digital Input - Generator circuit breaker closed*)
		bF07_DO_GCB_RUC : BOOL; (*Function 07 - Digital Output - GCB - Release undervoltage coil*)
		bF07_DO_Rel_Sync_Load : BOOL; (*Function 07 - Digital Output - Release synchronizing and load*)
		bF09_DI_ERV_INL1_Fan_Run : BOOL; (*Function 09 - Group 1 - Inlet air fan operating - Digital input*)
		bF09_DI_ERV_INL1_Lou_CL : BOOL; (*Function 09 - Group 1 - Inlet air louvre closed - Digital input*)
		bF09_DI_ERV_INL1_Lou_OP : BOOL; (*Function 09 - Group 1 - Inlet air louvre opened - Digital input*)
		bF09_DI_ERV_INL2_Fan_Run : BOOL; (*Function 09 - Group 2 - Inlet air fan operating - Digital input*)
		bF09_DI_ERV_INL2_Lou_CL : BOOL; (*Function 09 - Group 2 - Inlet air louvre closed - Digital input*)
		bF09_DI_ERV_INL2_Lou_OP : BOOL; (*Function 09 - Group 2 - Inlet air louvre opened - Digital input*)
		bF09_DI_ERV_INL3_Fan_Run : BOOL; (*Function 09 - Group 3 - Inlet air fan operating - Digital input*)
		bF09_DI_ERV_INL3_Lou_CL : BOOL; (*Function 09 - Group 3 - Inlet air louvre closed - Digital input*)
		bF09_DI_ERV_INL3_Lou_OP : BOOL; (*Function 09 - Group 3 - Inlet air louvre opened - Digital input*)
		bF09_DI_ERV_INL4_Fan_Run : BOOL; (*Function 09 - Group 4 - Inlet air fan operating - Digital input*)
		bF09_DI_ERV_INL4_Lou_CL : BOOL; (*Function 09 - Group 4 - Inlet air louvre closed - Digital input*)
		bF09_DI_ERV_INL4_Lou_OP : BOOL; (*Function 09 - Group 4 - Inlet air louvre opened - Digital input*)
		bF09_DI_ERV_INL5_Fan_Run : BOOL; (*Function 09 - Group 5 - Inlet air fan operating - Digital input*)
		bF09_DI_ERV_INL5_Lou_CL : BOOL; (*Function 09 - Group 5 - Inlet air louvre closed - Digital input*)
		bF09_DI_ERV_INL5_Lou_OP : BOOL; (*Function 09 - Group 5 - Inlet air louvre opened - Digital input*)
		bF09_DI_ERV_INL6_Fan_Run : BOOL; (*Function 09 - Group 6 - Inlet air fan operating - Digital input*)
		bF09_DI_ERV_INL6_Lou_CL : BOOL; (*Function 09 - Group 6 - Inlet air louvre closed - Digital input*)
		bF09_DI_ERV_INL6_Lou_OP : BOOL; (*Function 09 - Group 6 - Inlet air louvre opened - Digital input*)
		bF09_DI_ERV_OTL1_Lou_CL : BOOL; (*Function 09 - Group 1 - Outlet air louvre closed - Digital input*)
		bF09_DI_ERV_OTL1_Lou_OP : BOOL; (*Function 09 - Group 1 - Outlet air louvre opened - Digital input*)
		bF09_DI_ERV_OTL2_Lou_CL : BOOL; (*Function 09 - Group 2 - Outlet air louvre closed - Digital input*)
		bF09_DI_ERV_OTL2_Lou_OP : BOOL; (*Function 09 - Group 2 - Outlet air louvre opened - Digital input*)
		bF09_DI_ERV_OTL3_Lou_CL : BOOL; (*Function 09 - Group 3 - Outlet air louvre closed - Digital input*)
		bF09_DI_ERV_OTL3_Lou_OP : BOOL; (*Function 09 - Group 3 - Outlet air louvre opened - Digital input*)
		bF09_DI_ERV_OTL4_Lou_CL : BOOL; (*Function 09 - Group 4 - Outlet air louvre closed - Digital input*)
		bF09_DI_ERV_OTL4_Lou_OP : BOOL; (*Function 09 - Group 4 - Outlet air louvre opened - Digital input*)
		bF09_DI_ERV_OTL5_Lou_CL : BOOL; (*Function 09 - Group 5 - Outlet air louvre closed - Digital input*)
		bF09_DI_ERV_OTL5_Lou_OP : BOOL; (*Function 09 - Group 5 - Outlet air louvre opened - Digital input*)
		bF09_DI_ERV_OTL6_Lou_CL : BOOL; (*Function 09 - Group 6 - Outlet air louvre closed - Digital input*)
		bF09_DI_ERV_OTL6_Lou_OP : BOOL; (*Function 09 - Group 6 - Outlet air louvre opened - Digital input*)
		bF09_DI_ER_Door_CL : BOOL; (*Function 09 - Doors closed - Digital input*)
		bF09_ERV_ColdCountry : BOOL; (*Function 09 - Engine room ventilation - Cold country mode active*)
		bF10_Exist_EmStop_AUX : BOOL; (*Function 10 - Emergency stop push button exists - Auxiliaries control panel*)
		bF10_Exist_EmStop_EGAT : BOOL; (*Function 10 - Emergency stop push button exists - Exhaust gas after treatment control panel*)
		bF10_Exist_EmStop_ER1 : BOOL; (*Function 10 - Emergency stop push button exists - Engine room button 1*)
		bF10_Exist_EmStop_ER2 : BOOL; (*Function 10 - Emergency stop push button exists - Engine room button 2*)
		bF10_Exist_EmStop_ER3 : BOOL; (*Function 10 - Emergency stop push button exists - Engine room button 3*)
		bF10_Exist_EmStop_ER4 : BOOL; (*Function 10 - Emergency stop push button exists - Engine room button 4*)
		bF10_Exist_EmStop_EXT : BOOL; (*Function 10 - Emergency stop push button exists - External*)
		bF10_Exist_EmStop_IP : BOOL; (*Function 10 - Emergency stop push button exists - Interlock control panel*)
		bF10_Exist_EmStop_MC : BOOL; (*Function 10 - Emergency stop push button exists - Module control panel (+A/+MC)*)
		bF10_Exist_EmStop_MCP : BOOL; (*Function 10 - Emergency stop push button exists - Master control panel*)
		bF10_Exist_EmStop_PCGC : BOOL; (*Function 10 - Emergency stop push button exists - Prechamber gas compressor*)
		bF10_Exist_EmStop_TR : BOOL; (*Function 10 - Emergency stop push button exists - Thermal reactor control panel*)
		bF12_DO_DCGA_GV_Open : BOOL; (*Function 12 - Digital Output - Demand gas valves from DCGA*)
		bF12_DO_GV1_Open : BOOL; (*Function 12 - Digital Output - Demand gas valves from gas train 1*)
		bF12_DO_GV2_Open : BOOL; (*Function 12 - Digital Output - Demand gas valves from gas train 2*)
		bF12_DO_GV3_Open : BOOL; (*Function 12 - Digital Output - Demand gas valves from gas train 3*)
		bF12_DO_GV4_Open : BOOL; (*Function 12 - Digital Output - Demand gas valves from gas train 4*)
		bInfoSafeAppl_Ack : BOOL;
		bInfoSafeAppl_Exist : BOOL;
		bInfoSafeComm_Ack : BOOL;
		bInfoSafeComm_Exist : BOOL;
		bInfoStatus_FWExchanged : BOOL;
		bInfoStatus_SetupModeActive : BOOL;
		bInfoStatus_SKExchanged : BOOL;
		bInfoStatus_SNExchanged : BOOL;
		bInfo_Busy : BOOL;
		bInfo_Done : BOOL;
		bInfo_Error : BOOL;
		bLoadSafeOpt_Busy : BOOL;
		bLoadSafeOpt_Done : BOOL;
		bLoadSafeOpt_Error : BOOL;
		bParaSafe_DCGA_Exist : BOOL; (*From SafetyPLC - PARA [15196]: Gas train for decentral gas addition existing*)
		bParaSafe_ERV_ColdCountry_Active : BOOL; (*From SafetyPLC - PARA [15189]: Cold country mode active*)
		bParaSafe_ERV_Cust_Active : BOOL; (*From SafetyPLC - PARA [15188]: Customer room ventilation - Monitoring active*)
		bParaSafe_ER_Door_MonActive : BOOL; (*From SafetyPLC - PARA [15212]: Door switch - Monitoring active*)
		bParaSafe_FS_HWHT_Lo_Exist : BOOL; (*From SafetyPLC - PARA [15117]: High temperature heating water - Minimum flow switch available*)
		bParaSafe_FS_HWLT_Lo_Exist : BOOL; (*From SafetyPLC - PARA [15125]: Low temperature heating water - Minimum flow switch available*)
		bParaSafe_GT2_Exist : BOOL; (*From SafetyPLC - PARA [15082]: Gas train 2 existing*)
		bParaSafe_GT3_Exist : BOOL; (*From SafetyPLC - PARA [15083]: Gas train 3 existing*)
		bParaSafe_GT4_Exist : BOOL; (*From SafetyPLC - PARA [15103]: Gas train 4 existing*)
		bParaSafe_HWcirc_Cust_Exist : BOOL; (*From SafetyPLC - PARA [15108]: Customer heating water circuit - Monitoring active*)
		bParaSafe_LS_HWHT_Lo_Exist : BOOL; (*From SafetyPLC - PARA [15110]: High temperature heating water - Minimum level switch available*)
		bParaSafe_LS_HWLT_Lo_Exist : BOOL; (*From SafetyPLC - PARA [15118]: Low temperature heating water - Minimum level switch available*)
		bParaSafe_Pr_EG_sMonActive : BOOL; (*From SafetyPLC - PARA [15085]: Exhaust gas backpressure - Safety monitoring active*)
		bParaSafe_PS1_HWHT_Hi_Exist : BOOL; (*From SafetyPLC - PARA [15111]: High temperature heating water - Maximum pressure switch 1 available*)
		bParaSafe_PS1_HWHT_Lo_Exist : BOOL; (*From SafetyPLC - PARA [15113]: High temperature heating water - Minimum pressure switch 1 available*)
		bParaSafe_PS1_HWLT_Hi_Exist : BOOL; (*From SafetyPLC - PARA [15119]: Low temperature heating water - Maximum pressure switch 1 available*)
		bParaSafe_PS1_HWLT_Lo_Exist : BOOL; (*From SafetyPLC - PARA [15121]: Low temperature heating water - Minimum pressure switch 1 available*)
		bParaSafe_PS2_HWHT_Hi_Exist : BOOL; (*From SafetyPLC - PARA [15112]: High temperature heating water - Maximum pressure switch 2 available*)
		bParaSafe_PS2_HWHT_Lo_Exist : BOOL; (*From SafetyPLC - PARA [15114]: High temperature heating water - Minimum pressure switch 2 available*)
		bParaSafe_PS2_HWLT_Hi_Exist : BOOL; (*From SafetyPLC - PARA [15120]: Low temperature heating water - Maximum pressure switch 2 available*)
		bParaSafe_PS2_HWLT_Lo_Exist : BOOL; (*From SafetyPLC - PARA [15122]: Low temperature heating water - Minimum pressure switch 2 available*)
		bParaSafe_PS_HW_Lo_MuteActive : BOOL; (*From SafetyPLC - PARA [15109]: Muting heating water minimum pressure switches at engine standstill active*)
		bParaSafe_SafetyLoop_A2_Exist : BOOL; (*From SafetyPLC - PARA [15143]: Safety loop 2 in the module control panel existing*)
		bParaSafe_SysPurge_MonActive : BOOL; (*From SafetyPLC - PARA [15107]: System purge - Monitoring active*)
		bParaSafe_TS1_HWHT_Hi_Exist : BOOL; (*From SafetyPLC - PARA [15115]: High temperature heating water - Maximum temperature switch 1 available*)
		bParaSafe_TS1_HWLT_Hi_Exist : BOOL; (*From SafetyPLC - PARA [15123]: Low temperature heating water - Maximum temperature switch 1 available*)
		bParaSafe_TS2_HWHT_Hi_Exist : BOOL; (*From SafetyPLC - PARA [15116]: High temperature heating water - Maximum temperature switch 2 available*)
		bParaSafe_TS2_HWLT_Hi_Exist : BOOL; (*From SafetyPLC - PARA [15124]: Low temperature heating water - Maximum temperature switch 2 available*)
		bRead_CRC : BOOL; (*CRC readout of SafetyPLC is active*)
		bSafeModuleOK_101 : BOOL; (*Safe communication channel - Node 101 OK*)
		bSafeModuleOK_102 : BOOL; (*Safe communication channel - Node 102 OK*)
		bSafeModuleOK_103 : BOOL; (*Safe communication channel - Node 103 OK*)
		bSafeModuleOK_104 : BOOL; (*Safe communication channel - Node 104 OK*)
		bSafeModuleOK_105 : BOOL; (*Safe communication channel - Node 105 OK*)
		bSafeModuleOK_201 : BOOL; (*Safe communication channel - Node 201 OK*)
		bSafeModuleOK_202 : BOOL; (*Safe communication channel - Node 202 OK*)
		bSafeModuleOK_203 : BOOL; (*Safe communication channel - Node 203 OK*)
		bSafeModuleOK_204 : BOOL; (*Safe communication channel - Node 204 OK*)
		bSafeModuleOK_205 : BOOL; (*Safe communication channel - Node 205 OK*)
		bSafeModuleOK_206 : BOOL; (*Safe communication channel - Node 206 OK*)
		bSafeModuleOK_207 : BOOL; (*Safe communication channel - Node 207 OK*)
		bSafeModuleOK_208 : BOOL; (*Safe communication channel - Node 208 OK*)
		bSafeModuleOK_209 : BOOL; (*Safe communication channel - Node 209 OK*)
		bSafeModuleOK_210 : BOOL; (*Safe communication channel - Node 210 OK*)
		bSafeModuleOK_300 : BOOL; (*Safe communication channel - Node 300 OK*)
		bSafeModuleOK_301 : BOOL; (*Safe communication channel - Node 301 OK*)
		bSafeOUT_F01_N_DiffOK : BOOL; (*From SafetyPLC - Function 01 - Speed difference OK*)
		bSafeOUT_F01_N_Nom90 : BOOL; (*From SafetyPLC - Function 01 - Actual engine speed >= 90% of nominal speed*)
		bSafeOUT_F01_OK : BOOL; (*From SafetyPLC - Function 01 - Speed measurement OK*)
		bSafeOUT_F02_OK : BOOL; (*From SafetyPLC - Function 02 - Ignition is operating*)
		bSafeOUT_F02_OK_PC : BOOL; (*From SafetyPLC - Function 02 - Ignition plausibility check - OK*)
		bSafeOUT_F03_OK : BOOL; (*From SafetyPLC - Function 03 - Oil pressure MIN OK*)
		bSafeOUT_F03_Pr_EO_DiffOK : BOOL; (*From SafetyPLC - Function 03 - Oil pressure difference OK*)
		bSafeOUT_F04_OK : BOOL; (*From SafetyPLC - Function 04 - Oil pressure MAX OK*)
		bSafeOUT_F05_OK : BOOL; (*From SafetyPLC - Function 05 - Engine cooling water pressure MIN OK*)
		bSafeOUT_F05_Pr_ECW_DiffOK : BOOL; (*From SafetyPLC - Function 05 - Engine cooling water pressure difference OK*)
		bSafeOUT_F06_OK : BOOL; (*From SafetyPLC - Function 06 - Engine cooling water pressure MAX OK*)
		bSafeOUT_F07_GCB_RUC : BOOL; (*From SafetyPLC - Function 07 - GCB - Release undervoltage coil*)
		bSafeOUT_F07_GCB_RUC_PS : BOOL; (*From SafetyPLC - Function 07 - GCB - Release undervoltage coil - Physical state*)
		bSafeOUT_F07_OK : BOOL; (*From SafetyPLC - Function 07 - Grid disconnection OK*)
		bSafeOUT_F07_Rel_Sync_Load : BOOL; (*From SafetyPLC - Function 07 - Release synchronizing and load*)
		bSafeOUT_F07_Rel_Sync_Load_PS : BOOL; (*From SafetyPLC - Function 07 - Release synchronizing and load - Physical state*)
		bSafeOUT_F08_GenPrctTrip_OK : BOOL; (*From SafetyPLC - Function 08 - Generator protection trip OK*)
		bSafeOUT_F08_OlShortCirc_OK : BOOL; (*From SafetyPLC - Function 08 - Generator overload/short circuit OK*)
		bSafeOUT_F09_Cust_OK : BOOL; (*From SafetyPLC - Function 09 - Room ventilation operating*)
		bSafeOUT_F09_Cust_OK_PC : BOOL; (*From SafetyPLC - Function 09 - Room ventilation plausibility check OK*)
		bSafeOUT_F09_DI_ERV_Cust : BOOL; (*From SafetyPLC - Function 09 - Room ventilation operating - Digital input*)
		bSafeOUT_F09_Door_OK : BOOL; (*From SafetyPLC - Function 09 - Doors closed*)
		bSafeOUT_F09_INL1_Fan_OK : BOOL; (*From SafetyPLC - Function 09 - Group 1 - Inlet air fan operating*)
		bSafeOUT_F09_INL1_Fan_OK_PC : BOOL; (*From SafetyPLC - Function 09 - Group 1 - Inlet air fan plausibility check OK*)
		bSafeOUT_F09_INL1_Lou_OK : BOOL; (*From SafetyPLC - Function 09 - Group 1 - Inlet air louvre OK*)
		bSafeOUT_F09_INL1_Lou_OK_PC : BOOL; (*From SafetyPLC - Function 09 - Group 1 - Inlet air louvre plausibility check OK*)
		bSafeOUT_F09_INL2_Fan_OK : BOOL; (*From SafetyPLC - Function 09 - Group 2 - Inlet air fan operating*)
		bSafeOUT_F09_INL2_Fan_OK_PC : BOOL; (*From SafetyPLC - Function 09 - Group 2 - Inlet air fan plausibility check OK*)
		bSafeOUT_F09_INL2_Lou_OK : BOOL; (*From SafetyPLC - Function 09 - Group 2 - Inlet air louvre OK*)
		bSafeOUT_F09_INL2_Lou_OK_PC : BOOL; (*From SafetyPLC - Function 09 - Group 2 - Inlet air louvre plausibility check OK*)
		bSafeOUT_F09_INL3_Fan_OK : BOOL; (*From SafetyPLC - Function 09 - Group 3 - Inlet air fan operating*)
		bSafeOUT_F09_INL3_Fan_OK_PC : BOOL; (*From SafetyPLC - Function 09 - Group 3 - Inlet air fan plausibility check OK*)
		bSafeOUT_F09_INL3_Lou_OK : BOOL; (*From SafetyPLC - Function 09 - Group 3 - Inlet air louvre OK*)
		bSafeOUT_F09_INL3_Lou_OK_PC : BOOL; (*From SafetyPLC - Function 09 - Group 3 - Inlet air louvre plausibility check OK*)
		bSafeOUT_F09_INL4_Fan_OK : BOOL; (*From SafetyPLC - Function 09 - Group 4 - Inlet air fan operating*)
		bSafeOUT_F09_INL4_Fan_OK_PC : BOOL; (*From SafetyPLC - Function 09 - Group 4 - Inlet air fan plausibility check OK*)
		bSafeOUT_F09_INL4_Lou_OK : BOOL; (*From SafetyPLC - Function 09 - Group 4 - Inlet air louvre OK*)
		bSafeOUT_F09_INL4_Lou_OK_PC : BOOL; (*From SafetyPLC - Function 09 - Group 4 - Inlet air louvre plausibility check OK*)
		bSafeOUT_F09_INL5_Fan_OK : BOOL; (*From SafetyPLC - Function 09 - Group 5 - Inlet air fan operating*)
		bSafeOUT_F09_INL5_Fan_OK_PC : BOOL; (*From SafetyPLC - Function 09 - Group 5 - Inlet air fan plausibility check OK*)
		bSafeOUT_F09_INL5_Lou_OK : BOOL; (*From SafetyPLC - Function 09 - Group 5 - Inlet air louvre OK*)
		bSafeOUT_F09_INL5_Lou_OK_PC : BOOL; (*From SafetyPLC - Function 09 - Group 5 - Inlet air louvre plausibility check OK*)
		bSafeOUT_F09_INL6_Fan_OK : BOOL; (*From SafetyPLC - Function 09 - Group 6 - Inlet air fan operating*)
		bSafeOUT_F09_INL6_Fan_OK_PC : BOOL; (*From SafetyPLC - Function 09 - Group 6 - Inlet air fan plausibility check OK*)
		bSafeOUT_F09_INL6_Lou_OK : BOOL; (*From SafetyPLC - Function 09 - Group 6 - Inlet air louvre OK*)
		bSafeOUT_F09_INL6_Lou_OK_PC : BOOL; (*From SafetyPLC - Function 09 - Group 6 - Inlet air louvre plausibility check OK*)
		bSafeOUT_F09_OTL1_Lou_OK : BOOL; (*From SafetyPLC - Function 09 - Group 1 - Outlet air louvre OK*)
		bSafeOUT_F09_OTL1_Lou_OK_PC : BOOL; (*From SafetyPLC - Function 09 - Group 1 - Outlet air louvre plausibility check OK*)
		bSafeOUT_F09_OTL2_Lou_OK : BOOL; (*From SafetyPLC - Function 09 - Group 2 - Outlet air louvre OK*)
		bSafeOUT_F09_OTL2_Lou_OK_PC : BOOL; (*From SafetyPLC - Function 09 - Group 2 - Outlet air louvre plausibility check OK*)
		bSafeOUT_F09_OTL3_Lou_OK : BOOL; (*From SafetyPLC - Function 09 - Group 3 - Outlet air louvre OK*)
		bSafeOUT_F09_OTL3_Lou_OK_PC : BOOL; (*From SafetyPLC - Function 09 - Group 3 - Outlet air louvre plausibility check OK*)
		bSafeOUT_F09_OTL4_Lou_OK : BOOL; (*From SafetyPLC - Function 09 - Group 4 - Outlet air louvre OK*)
		bSafeOUT_F09_OTL4_Lou_OK_PC : BOOL; (*From SafetyPLC - Function 09 - Group 4 - Outlet air louvre plausibility check OK*)
		bSafeOUT_F09_OTL5_Lou_OK : BOOL; (*From SafetyPLC - Function 09 - Group 5 - Outlet air louvre OK*)
		bSafeOUT_F09_OTL5_Lou_OK_PC : BOOL; (*From SafetyPLC - Function 09 - Group 5 - Outlet air louvre plausibility check OK*)
		bSafeOUT_F09_OTL6_Lou_OK : BOOL; (*From SafetyPLC - Function 09 - Group 6 - Outlet air louvre OK*)
		bSafeOUT_F09_OTL6_Lou_OK_PC : BOOL; (*From SafetyPLC - Function 09 - Group 6 - Outlet air louvre plausibility check OK*)
		bSafeOUT_F10_DO_EmStop : BOOL; (*From SafetyPLC - Function 10 - DO Emergency stop signalling*)
		bSafeOUT_F10_DO_EmStop_PS : BOOL; (*From SafetyPLC - Function 10 - DO Emergency stop signalling - Physical state*)
		bSafeOUT_F10_EmStop_M_OK : BOOL; (*From SafetyPLC - Function 10 - Emergency stop push button - Module interface panel*)
		bSafeOUT_F10_EmStop_OK : BOOL; (*From SafetyPLC - Function 10 - Emergency stop push button*)
		bSafeOUT_F11_OK : BOOL; (*From SafetyPLC - Function 11 - RESERVE*)
		bSafeOUT_F11_SafetyLoop_A1_OK : BOOL; (*From SafetyPLC - Function 11 - Safety loop 1 - module control panel OK*)
		bSafeOUT_F11_SafetyLoop_A2_OK : BOOL; (*From SafetyPLC - Function 11 - Safety loop 2 - module control panel OK*)
		bSafeOUT_F11_SafetyLoop_M_OK : BOOL; (*From SafetyPLC - Function 11 - Safety loop - module interface panel OK*)
		bSafeOUT_F12_DCGA_OK : BOOL; (*From SafetyPLC - Function 12 - Gas supply interruption OK - DCGA (Decentral gas addition)*)
		bSafeOUT_F12_DCGA_SD_Dem : BOOL; (*From SafetyPLC - Function 12 - Demand gas safety device - DCGA*)
		bSafeOUT_F12_DCGA_SD_Dem_PS : BOOL; (*From SafetyPLC - Function 12 - Demand gas safety device - DCGA - Physical state*)
		bSafeOUT_F12_DI_DCGA_SafeDevOK : BOOL; (*From SafetyPLC - Function 12 - Digital Input - Gas safety device OK - DCGA*)
		bSafeOUT_F12_DI_GT1_SafeDevOK : BOOL; (*From SafetyPLC - Function 12 - Digital Input - Gas safety device OK - Gastrain 1*)
		bSafeOUT_F12_DI_GT2_SafeDevOK : BOOL; (*From SafetyPLC - Function 12 - Digital Input - Gas safety device OK - Gastrain 2*)
		bSafeOUT_F12_DI_GT3_SafeDevOK : BOOL; (*From SafetyPLC - Function 12 - Digital Input - Gas safety device OK - Gastrain 3*)
		bSafeOUT_F12_DI_GT4_SafeDevOK : BOOL; (*From SafetyPLC - Function 12 - Digital Input - Gas safety device OK - Gastrain 4*)
		bSafeOUT_F12_GT1_OK : BOOL; (*From SafetyPLC - Function 12 - Gas supply interruption OK - Gas train 1*)
		bSafeOUT_F12_GT1_SD_Dem : BOOL; (*From SafetyPLC - Function 12 - Demand gas safety device - Gastrain 1*)
		bSafeOUT_F12_GT1_SD_Dem_PS : BOOL; (*From SafetyPLC - Function 12 - Demand gas safety device - Gastrain 1 - Physical state*)
		bSafeOUT_F12_GT2_OK : BOOL; (*From SafetyPLC - Function 12 - Gas supply interruption OK - Gas train 2*)
		bSafeOUT_F12_GT2_SD_Dem : BOOL; (*From SafetyPLC - Function 12 - Demand gas safety device - Gastrain 2*)
		bSafeOUT_F12_GT2_SD_Dem_PS : BOOL; (*From SafetyPLC - Function 12 - Demand gas safety device - Gastrain 2 - Physical state*)
		bSafeOUT_F12_GT3_OK : BOOL; (*From SafetyPLC - Function 12 - Gas supply interruption OK - Gas train 3*)
		bSafeOUT_F12_GT3_SD_Dem : BOOL; (*From SafetyPLC - Function 12 - Demand gas safety device - Gastrain 3*)
		bSafeOUT_F12_GT3_SD_Dem_PS : BOOL; (*From SafetyPLC - Function 12 - Demand gas safety device - Gastrain 3 - Physical state*)
		bSafeOUT_F12_GT4_OK : BOOL; (*From SafetyPLC - Function 12 - Gas supply interruption OK - Gas train 4*)
		bSafeOUT_F12_GT4_SD_Dem : BOOL; (*From SafetyPLC - Function 12 - Demand gas safety device - Gastrain 4*)
		bSafeOUT_F12_GT4_SD_Dem_PS : BOOL; (*From SafetyPLC - Function 12 - Demand gas safety device - Gastrain 4 - Physical state*)
		bSafeOUT_F12_Rel_GV1 : BOOL; (*From SafetyPLC - Function 12 - Gas valves from gas train 1 released*)
		bSafeOUT_F12_Rel_GV1a_PS : BOOL; (*From SafetyPLC - Function 12 - Gas valve 1a - Physical state*)
		bSafeOUT_F12_Rel_GV1b_PS : BOOL; (*From SafetyPLC - Function 12 - Gas valve 1b - Physical state*)
		bSafeOUT_F12_Rel_GV2 : BOOL; (*From SafetyPLC - Function 12 - Gas valves from gas train 2 released*)
		bSafeOUT_F12_Rel_GV2a_PS : BOOL; (*From SafetyPLC - Function 12 - Gas valve 2a - Physical state*)
		bSafeOUT_F12_Rel_GV2b_PS : BOOL; (*From SafetyPLC - Function 12 - Gas valve 2b - Physical state*)
		bSafeOUT_F12_Rel_GV3 : BOOL; (*From SafetyPLC - Function 12 - Gas valves from gas train 3 released*)
		bSafeOUT_F12_Rel_GV3a_PS : BOOL; (*From SafetyPLC - Function 12 - Gas valve 3a - Physical state*)
		bSafeOUT_F12_Rel_GV3b_PS : BOOL; (*From SafetyPLC - Function 12 - Gas valve 3b - Physical state*)
		bSafeOUT_F12_Rel_GV4 : BOOL; (*From SafetyPLC - Function 12 - Gas valves from gas train 4 released*)
		bSafeOUT_F12_Rel_GV4a_PS : BOOL; (*From SafetyPLC - Function 12 - Gas valve 4a - Physical state*)
		bSafeOUT_F12_Rel_GV4b_PS : BOOL; (*From SafetyPLC - Function 12 - Gas valve 4b - Physical state*)
		bSafeOUT_F12_Rel_GVa_DCGA_PS : BOOL; (*From SafetyPLC - Function 12 - Gas valve a for DCGA - Physical state*)
		bSafeOUT_F12_Rel_GVb_DCGA_PS : BOOL; (*From SafetyPLC - Function 12 - Gas valve b for DCGA - Physical state*)
		bSafeOUT_F12_Rel_GV_DCGA : BOOL; (*From SafetyPLC - Function 12 - Gas valves from DCGA released*)
		bSafeOUT_F16_DI_ScavFlapClosed : BOOL; (*From SafetyPLC - Function 20 - Scavenging flap closed OK*)
		bSafeOUT_F16_ScavFlapPos_OK : BOOL; (*From SafetyPLC - Function 20 - Scavenging flap position OK*)
		bSafeOUT_F16_ScavFlapPos_OK_PC : BOOL; (*From SafetyPLC - Function 20 - Scavenging flap position - plausibility check  OK*)
		bSafeOUT_F16_TS_ScavFlap_OK : BOOL; (*From SafetyPLC - Function 20 - Scavenging flap temperature switch  OK*)
		bSafeOUT_F20_FS_HWHT_Lo_DI : BOOL; (*From SafetyPLC - Function 20 - High temperature heating water flow minimum - DI OK*)
		bSafeOUT_F20_FS_HWHT_Lo_OK : BOOL; (*From SafetyPLC - Function 20 - High temperature heating water flow minimum OK*)
		bSafeOUT_F20_FS_HWHT_Lo_OK_PC : BOOL; (*From SafetyPLC - Function 20 - High temperature heating water flow minimum - plausibility check OK*)
		bSafeOUT_F20_FS_HWLT_Lo_DI : BOOL; (*From SafetyPLC - Function 20 - Low temperature heating water flow minimum - DI OK*)
		bSafeOUT_F20_FS_HWLT_Lo_OK : BOOL; (*From SafetyPLC - Function 20 - Low temperature heating water flow minimum OK*)
		bSafeOUT_F20_FS_HWLT_Lo_OK_PC : BOOL; (*From SafetyPLC - Function 20 - Low temperature heating water flow minimum - plausibility check OK*)
		bSafeOUT_F20_HWcirc_Cust_OK : BOOL; (*From SafetyPLC - Function 20 - Customer heating water circuit OK*)
		bSafeOUT_F20_LS_HWHT_Lo_OK : BOOL; (*From SafetyPLC - Function 20 - High temperature heating water level minimum OK*)
		bSafeOUT_F20_LS_HWLT_Lo_OK : BOOL; (*From SafetyPLC - Function 20 - Low temperature heating water level minimum OK*)
		bSafeOUT_F20_PS1_HWHT_Hi_OK : BOOL; (*From SafetyPLC - Function 20 - High temperature heating water pressure 1 maximum OK*)
		bSafeOUT_F20_PS1_HWHT_Lo_DI : BOOL; (*From SafetyPLC - Function 20 - High temperature heating water pressure 1 minimum - DI OK*)
		bSafeOUT_F20_PS1_HWHT_Lo_OK : BOOL; (*From SafetyPLC - Function 20 - High temperature heating water pressure 1 minimum OK*)
		bSafeOUT_F20_PS1_HWLT_Hi_OK : BOOL; (*From SafetyPLC - Function 20 - Low temperature heating water pressure 1 maximum OK*)
		bSafeOUT_F20_PS1_HWLT_Lo_DI : BOOL; (*From SafetyPLC - Function 20 - Low temperature heating water pressure 1 minimum - DI OK*)
		bSafeOUT_F20_PS1_HWLT_Lo_OK : BOOL; (*From SafetyPLC - Function 20 - Low temperature heating water pressure 1 minimum OK*)
		bSafeOUT_F20_PS2_HWHT_Hi_OK : BOOL; (*From SafetyPLC - Function 20 - High temperature heating water pressure 2 maximum OK*)
		bSafeOUT_F20_PS2_HWHT_Lo_DI : BOOL; (*From SafetyPLC - Function 20 - High temperature heating water pressure 2 minimum - DI OK*)
		bSafeOUT_F20_PS2_HWHT_Lo_OK : BOOL; (*From SafetyPLC - Function 20 - High temperature heating water pressure 2 minimum OK*)
		bSafeOUT_F20_PS2_HWLT_Hi_OK : BOOL; (*From SafetyPLC - Function 20 - Low temperature heating water pressure 2 maximum OK*)
		bSafeOUT_F20_PS2_HWLT_Lo_DI : BOOL; (*From SafetyPLC - Function 20 - Low temperature heating water pressure 2 minimum - DI OK*)
		bSafeOUT_F20_PS2_HWLT_Lo_OK : BOOL; (*From SafetyPLC - Function 20 - Low temperature heating water pressure 2 minimum OK*)
		bSafeOUT_F20_TS1_HWHT_Hi_OK : BOOL; (*From SafetyPLC - Function 20 - High temperature heating water temperature 1 maximum OK*)
		bSafeOUT_F20_TS1_HWLT_Hi_OK : BOOL; (*From SafetyPLC - Function 20 - Low temperature heating water temperature 1 maximum OK*)
		bSafeOUT_F20_TS2_HWHT_Hi_OK : BOOL; (*From SafetyPLC - Function 20 - High temperature heating water temperature 2 maximum OK*)
		bSafeOUT_F20_TS2_HWLT_Hi_OK : BOOL; (*From SafetyPLC - Function 20 - Low temperature heating water temperature 2 maximum OK*)
		bSafeOUT_F21_Pr_EG_Hi_OK : BOOL; (*From SafetyPLC - Function 20 - Exhaust gas backpressure high OK*)
		bSafeOUT_F99_Rel_SF_OK : BOOL; (*From SafetyPLC - Function 99 - Release safety functions OK*)
		bSafeOUT_F99_Rel_SF_OK_A_PS : BOOL; (*From SafetyPLC - Function 99 - Release safety functions - Module control panel - Physical state*)
		bSafeOUT_F99_Rel_SF_OK_M_PS : BOOL; (*From SafetyPLC - Function 99 - Release safety functions - Module interface panel - Physical state*)
		bSafeOUT_SafetyPLC_Exist : BOOL; (*From SafetyPLC - IF hardware SL8100 exist -> SafetyPLC exist*)
		bSaveSafeOpt_Busy : BOOL;
		bSaveSafeOpt_Done : BOOL;
		bSaveSafeOpt_Error : BOOL;
		bSetSafeNodeAvail_Busy : BOOL;
		bSetSafeNodeAvail_Done : BOOL;
		bSetSafeNodeAvail_Error : BOOL;
		bSetSafeOptBool_Busy : BOOL;
		bSetSafeOptBool_Done : BOOL;
		bSetSafeOptBool_Error : BOOL;
		bSetSafeOptInt_Busy : BOOL;
		bSetSafeOptInt_Done : BOOL;
		bSetSafeOptInt_Error : BOOL;
		bTransfer_Busy : BOOL;
		bTransfer_Done : BOOL;
		bTransfer_Error : BOOL;
		iComError : DINT; (*Commissioning - Error*)
		iCompletion_StatusID : INT;
		iComStep : StepEnum; (*Commissioning - Step*)
		iConnect_PermLevel : INT;
		iConnect_SafeDomainID : INT;
		iConnect_StatusID : INT;
		iConnect_UDID_high : INT;
		iConnect_UDID_low : INT;
		iControl_StatusID : INT;
		iDownloadStep : INT;
		iExchange_StatusID : INT;
		iInfoSafeComm_CRC : INT;
		iInfoStatus_NoFWExchanged : INT;
		iInfoStatus_NoSafeNODEs : INT;
		iInfoStatus_NoSNExchanged : INT;
		iInfoStatus_OpModeState : INT;
		iInfoStatus_SafeComUnused : INT;
		iInfoStatus_SafeNodesState : INT;
		iInfoStatus_SafeOSState : INT;
		iInfoStatus_SystemState : INT;
		iInfo_StatusID : INT;
		iLoadSafeOpt_CRC : INT;
		iLoadSafeOpt_StatusID : INT;
		iNode_sPLC : UINT; (*SafetyPLC node*)
		iParaSafe_Eng_Motortype : INT; (*From SafetyPLC - PARA [15084]: Motortype*)
		iParaSafe_NrMaxErr_ERV_INL_Fan : INT; (*From SafetyPLC - PARA [15193]: Maximum allowed number of failed inlet air fans*)
		iParaSafe_NrMaxErr_ERV_INL_Lou : INT; (*From SafetyPLC - PARA [15194]: Maximum allowed number of failed inlet air louvres*)
		iParaSafe_NrMaxErr_ERV_OTL_Lou : INT; (*From SafetyPLC - PARA [15195]: Maximum allowed number of failed outlet air louvres*)
		iParaSafe_Nr_ERV_INL_Fan : INT; (*From SafetyPLC - PARA [15190]: Number of inlet air fans*)
		iParaSafe_Nr_ERV_INL_Lou : INT; (*From SafetyPLC - PARA [15191]: Number of inlet air louvres*)
		iParaSafe_Nr_ERV_OTL_Lou : INT; (*From SafetyPLC - PARA [15192]: Number of outlet air louvres*)
		iSafeOUT_F09_Nr_PC_NotDone : INT; (*From SafetyPLC - Function 09 - Number of plausibility checks not performed*)
		iSafeOUT_FwVers_sPLC : UDINT; (*From SafetyPLC - Actual firmware version*)
		iSaveSafeOpt_CRC : INT;
		iSaveSafeOpt_StatusID : INT;
		iSetSafeNodeAvail_StatusID : INT;
		iSetSafeNodeAvail_Value : INT;
		iSetSafeOptBool_StatusID : INT;
		iSetSafeOptInt_StatusID : INT;
		iSetSafeOptInt_Value : INT;
		iTransfer_Progress : INT;
		iTransfer_StatusID : INT;
		rParaSafe_DPr_ECWP_LoLo : REAL; (*From SafetyPLC - PARA [15104]: Engine cooling water pump - Difference pressure minimum [bar]*)
		rParaSafe_N_EngAct_HiHi_Diff : REAL; (*From SafetyPLC - PARA [15086]: Speed - Maximum deviation to ignition speed [rpm]*)
		rParaSafe_N_EngNom : REAL; (*From SafetyPLC - PARA [15087]: Speed - Nominal speed [rpm]*)
		rParaSafe_N_Pr_EO_LoLo_Lim1 : REAL; (*From SafetyPLC - PARA [15088]: Oil pressure - Minimum - Speed point 1 [rpm]*)
		rParaSafe_N_Pr_EO_LoLo_Lim2 : REAL; (*From SafetyPLC - PARA [15089]: Oil pressure - Minimum - Speed point 2 [rpm]*)
		rParaSafe_Pr_ECWaP_HiHi : REAL; (*From SafetyPLC - PARA [15093]: Engine cooling water pressure after pump - Maximum [mbar]*)
		rParaSafe_Pr_ECW_HiHi_Check : REAL; (*From SafetyPLC - PARA [15090]: Engine cooling water pressure - Maximum (sensor drift) [mbar]*)
		rParaSafe_Pr_ECW_HiHi_Diff : REAL; (*From SafetyPLC - PARA [15091]: Engine cooling water pressure - Maximum deviation between the sensors [mbar]*)
		rParaSafe_Pr_ECW_LoLo : REAL; (*From SafetyPLC - PARA [15092]: Engine cooling water pressure - Minimum [mbar]*)
		rParaSafe_Pr_EOaP_Diff_EngStop : REAL; (*From SafetyPLC - PARA [15100]: Oil pressure after pump - Minimum difference to standstill [mbar]*)
		rParaSafe_Pr_EOaP_HiHi : REAL; (*From SafetyPLC - PARA [15101]: Oil pressure after pump - Maximum [mbar]*)
		rParaSafe_Pr_EOaP_HiHi_EngStop : REAL; (*From SafetyPLC - PARA [15102]: Oil pressure after pump - Maximum at standstill [mbar]*)
		rParaSafe_Pr_EO_Diff_EngStop : REAL; (*From SafetyPLC - PARA [15094]: Oil pressure - Minimum difference to standstill [mbar]*)
		rParaSafe_Pr_EO_HiHi_Check : REAL; (*From SafetyPLC - PARA [15095]: Oil pressure - Maximum (sensor drift) [mbar]*)
		rParaSafe_Pr_EO_HiHi_Diff : REAL; (*From SafetyPLC - PARA [15096]: Oil pressure - Maximum deviation between the sensors [mbar]*)
		rParaSafe_Pr_EO_HiHi_EngStop : REAL; (*From SafetyPLC - PARA [15097]: Oil pressure - Maximum at standstill [mbar]*)
		rParaSafe_Pr_EO_LoLo_LimN1 : REAL; (*From SafetyPLC - PARA [15098]: Oil pressure - Minimum at speed point 1 [mbar]*)
		rParaSafe_Pr_EO_LoLo_LimN2 : REAL; (*From SafetyPLC - PARA [15099]: Oil pressure - Minimum at speed point 2 [mbar]*)
		rParaSafe_Vol_SysPurge_MinAir : REAL; (*From SafetyPLC - PARA [15106]: System purge - Minimum air volume [l]*)
		rParaSafe_Vol_SysPurge_Stroke : REAL; (*From SafetyPLC - PARA [15105]: System purge - Stroke volume per crankshaft turn [l/turn]*)
		rSafeOUT_F01_N_EngAct : REAL; (*From SafetyPLC - Function 01 - Actual engine speed [rpm]*)
		rSafeOUT_F01_N_EngAct_Diff : REAL; (*From SafetyPLC - Function 01 - Speed difference [rpm]*)
		rSafeOUT_F03_Pr_EO : REAL; (*From SafetyPLC - Function 03 - Actual oil pressure at last lubrication point [bar]*)
		rSafeOUT_F03_Pr_EO_Diff : REAL; (*From SafetyPLC - Function 03 - Oil pressure difference [bar]*)
		rSafeOUT_F03_Pr_EO_Standstill : REAL; (*From SafetyPLC - Function 03 - Oil pressure at last lubrication point - At standstill [bar]*)
		rSafeOUT_F04_Pr_EOaP : REAL; (*From SafetyPLC - Function 04 - Actual oil pressure after pump [bar]*)
		rSafeOUT_F04_Pr_EOaP_Standstill : REAL; (*From SafetyPLC - Function 04 - Oil pressure after pump - At standstill [bar]*)
		rSafeOUT_F05_Pr_ECW : REAL; (*From SafetyPLC - Function 05 - Actual engine cooling water pressure [bar]*)
		rSafeOUT_F05_Pr_ECW_Diff : REAL; (*From SafetyPLC - Function 05 - Engine cooling water pressure difference [bar]*)
		rSafeOUT_F06_Pr_ECWaP : REAL; (*From SafetyPLC - Function 06 - Actual engine cooling water pressure after pump [bar]*)
		szConnect_CurrentUser : STRING[80];
		szInfoSafeAppl_CRC : STRING[80]; (*From SafetyPLC - CRC*)
		szInfoSafeAppl_Name : STRING[80]; (*From SafetyPLC - Application name*)
		szInfoSafeAppl_TimeStamp : STRING[80]; (*From SafetyPLC - Time stamp*)
		szInfoSafeAppl_UserName : STRING[80]; (*From SafetyPLC - User name*)
		szInfoSafeComm_Name : STRING[80];
		szInfoSafeComm_TimeStamp : STRING[80];
		szInfoSafeComm_UserName : STRING[80];
		szSafeOUT_F09_CRC : STRING[80]; (*From SafetyPLC - Function 09 - CRC for ventilation*)
		szSafeOUT_F20_CRC : STRING[80]; (*From SafetyPLC - Function 20 - CRC for heating water*)
		szSetSafeNodeAvail_OptionID : STRING[80];
		szSetSafeOptBool_OptionID : STRING[80];
		szSetSafeOptInt_OptionID : STRING[80];
		tiSafeOUT_F01_N_Nom90_10s_ET : TIME; (*From SafetyPLC - Function 01 - Speed >= 90% of nominal speed - Elipsed time*)
		tiSafeOUT_F01_SDC_30s_ET : TIME; (*From SafetyPLC - Function 01 - Speed difference check - Elipsed time*)
		tiSafeOUT_F01_Standstill_1m_ET : TIME; (*From SafetyPLC - Function 01 - Speed < 80rpm - Elipsed time*)
		tiSafeOUT_F03_Pr_EO_Fr_1m_ET : TIME; (*From SafetyPLC - Function 03 - Oil pressure frozen - Elipsed time*)
		tiSafeOUT_F04_EO_PumpsOff_2m_ET : TIME; (*From SafetyPLC - Function 04 - Oil pumps off for 120s - Elipsed time*)
		tiSafeOUT_F04_Pr_EOaP_Fr_1m_ET : TIME; (*From SafetyPLC - Function 04 - Oil pressure after pump frozen - Elipsed time*)
		tiSafeOUT_F05_Pr_ECW_Fr_1m_ET : TIME; (*From SafetyPLC - Function 05 - Engine cooling water pressure frozen - Elipsed time*)
		tiSafeOUT_F06_ECW_PumpsOff_2m_ET : TIME; (*From SafetyPLC - Function 06 - Engine cooling water pumps off for 120s - Elipsed time*)
		tiSafeOUT_F06_Pr_ECWaP_Fr_1m_ET : TIME; (*From SafetyPLC - Function 06 - Engine cooling water pressure after pump frozen - Elipsed time*)
		tiSafeOUT_F07_GCB_On_10s_ET : TIME; (*From SafetyPLC - Function 07 - Generator circuit breaker ON for 10s - Elipsed time*)
		tiSafeOUT_F07_GCB_On_60s_ET : TIME; (*From SafetyPLC - Function 07 - Generator circuit breaker ON for 60s - Elipsed time*)
		tiSafeOUT_F09_Cust_OK_15s_ET : TIME; (*From SafetyPLC - Function 09 - Room ventilation not operating - Elapsed time*)
		tiSafeOUT_F09_Cust_PC_ET : TIME; (*From SafetyPLC - Function 09 - Room ventilation plausibility check - Elapsed time*)
		tiSafeOUT_F09_Door_OK_15s_ET : TIME; (*From SafetyPLC - Function 09 - Doors not closed - Elapsed time*)
		tiSafeOUT_F09_INL1_Fan_OK_1m_ET : TIME; (*From SafetyPLC - Function 09 - Group 1 - Inlet air fan not operating - Elapsed time*)
		tiSafeOUT_F09_INL1_Lou_OK_1m_ET : TIME; (*From SafetyPLC - Function 09 - Group 1 - Inlet air louvre not OK - Elapsed time*)
		tiSafeOUT_F09_INL2_Fan_OK_1m_ET : TIME; (*From SafetyPLC - Function 09 - Group 2 - Inlet air fan not operating - Elapsed time*)
		tiSafeOUT_F09_INL2_Lou_OK_1m_ET : TIME; (*From SafetyPLC - Function 09 - Group 2 - Inlet air louvre not OK - Elapsed time*)
		tiSafeOUT_F09_INL3_Fan_OK_1m_ET : TIME; (*From SafetyPLC - Function 09 - Group 3 - Inlet air fan not operating - Elapsed time*)
		tiSafeOUT_F09_INL3_Lou_OK_1m_ET : TIME; (*From SafetyPLC - Function 09 - Group 3 - Inlet air louvre not OK - Elapsed time*)
		tiSafeOUT_F09_INL4_Fan_OK_1m_ET : TIME; (*From SafetyPLC - Function 09 - Group 4 - Inlet air fan not operating - Elapsed time*)
		tiSafeOUT_F09_INL4_Lou_OK_1m_ET : TIME; (*From SafetyPLC - Function 09 - Group 4 - Inlet air louvre not OK - Elapsed time*)
		tiSafeOUT_F09_INL5_Fan_OK_1m_ET : TIME; (*From SafetyPLC - Function 09 - Group 5 - Inlet air fan not operating - Elapsed time*)
		tiSafeOUT_F09_INL5_Lou_OK_1m_ET : TIME; (*From SafetyPLC - Function 09 - Group 5 - Inlet air louvre not OK - Elapsed time*)
		tiSafeOUT_F09_INL6_Fan_OK_1m_ET : TIME; (*From SafetyPLC - Function 09 - Group 6 - Inlet air fan not operating - Elapsed time*)
		tiSafeOUT_F09_INL6_Lou_OK_1m_ET : TIME; (*From SafetyPLC - Function 09 - Group 6 - Inlet air louvre not OK - Elapsed time*)
		tiSafeOUT_F09_OTL1_Lou_OK_1m_ET : TIME; (*From SafetyPLC - Function 09 - Group 1 - Outlet air louvre not OK - Elapsed time*)
		tiSafeOUT_F09_OTL2_Lou_OK_1m_ET : TIME; (*From SafetyPLC - Function 09 - Group 2 - Outlet air louvre not OK - Elapsed time*)
		tiSafeOUT_F09_OTL3_Lou_OK_1m_ET : TIME; (*From SafetyPLC - Function 09 - Group 3 - Outlet air louvre not OK - Elapsed time*)
		tiSafeOUT_F09_OTL4_Lou_OK_1m_ET : TIME; (*From SafetyPLC - Function 09 - Group 4 - Outlet air louvre not OK - Elapsed time*)
		tiSafeOUT_F09_OTL5_Lou_OK_1m_ET : TIME; (*From SafetyPLC - Function 09 - Group 5 - Outlet air louvre not OK - Elapsed time*)
		tiSafeOUT_F09_OTL6_Lou_OK_1m_ET : TIME; (*From SafetyPLC - Function 09 - Group 6 - Outlet air louvre not OK - Elapsed time*)
		tiSafeOUT_F12_DCGA_LC_130s_ET : TIME; (*From SafetyPLC - Function 12 - DCGA - Gas leakage check 130s - Elipsed time*)
		tiSafeOUT_F12_GT1_LC_130s_ET : TIME; (*From SafetyPLC - Function 12 - Gas train 1 - Gas leakage check 130s - Elipsed time*)
		tiSafeOUT_F12_GT2_LC_130s_ET : TIME; (*From SafetyPLC - Function 12 - Gas train 2 - Gas leakage check 130s - Elipsed time*)
		tiSafeOUT_F12_GT3_LC_130s_ET : TIME; (*From SafetyPLC - Function 12 - Gas train 3 - Gas leakage check 130s - Elipsed time*)
		tiSafeOUT_F12_GT4_LC_130s_ET : TIME; (*From SafetyPLC - Function 12 - Gas train 4 - Gas leakage check 130s - Elipsed time*)
		tiSafeOUT_F12_GV_Open_60s_ET : TIME; (*From SafetyPLC - Function 12 - Gas valves open for 60s - Elipsed time*)
		tiSafeOUT_F16_ScavFlapPos_PC_ET : TIME; (*From SafetyPLC - Function 20 - Scavenging flap position - plausibility check - Elipsed time OK*)
		tiSafeOUT_F20_FS_HWHT_Lo_OK_ET : TIME; (*From SafetyPLC - Function 20 - High temperature heating water flow minimum - Elipsed time OK*)
		tiSafeOUT_F20_FS_HWHT_Lo_PC_ET : TIME; (*From SafetyPLC - Function 20 - High temperature heating water flow minimum - plausibility check - Elipsed time OK*)
		tiSafeOUT_F20_FS_HWLT_Lo_OK_ET : TIME; (*From SafetyPLC - Function 20 - Low temperature heating water flow minimum - Elipsed time OK*)
		tiSafeOUT_F20_FS_HWLT_Lo_PC_ET : TIME; (*From SafetyPLC - Function 20 - Low temperature heating water flow minimum - plausibility check - Elipsed time OK*)
		tiSafeOUT_F20_PS1_HWHT_Lo_OK_ET : TIME; (*From SafetyPLC - Function 20 - High temperature heating water pressure 1 minimum - Elipsed time OK*)
		tiSafeOUT_F20_PS1_HWLT_Lo_OK_ET : TIME; (*From SafetyPLC - Function 20 - Low temperature heating water pressure 1 minimum - Elipsed time OK*)
		tiSafeOUT_F20_PS2_HWHT_Lo_OK_ET : TIME; (*From SafetyPLC - Function 20 - High temperature heating water pressure 2 minimum - Elipsed time OK*)
		tiSafeOUT_F20_PS2_HWLT_Lo_OK_ET : TIME; (*From SafetyPLC - Function 20 - Low temperature heating water pressure 2 minimum - Elipsed time OK*)
	END_STRUCT;
	VIS2MM_sPLC_struct : 	STRUCT
		bComDataCorrect : BOOL; (*Commissioning - Acknowledge data read from SafeDOMAIN is correct*)
		bComStartCmd : BOOL; (*Commissioning - Start command*)
		bConnect_UDID_Ack : BOOL;
		bControl_Execute_Dem : BOOL;
		bControl_Reboot_sPLC_Dem : BOOL; (*Demand - Reboot of SafetyPLC*)
		bExchange_Ack : BOOL;
		szConnect_UserName : STRING[80]; (*User Name*)
		szConnect_UserPassword : STRING[80]; (*User Password*)
	END_STRUCT;
	StepEnum :
		( (*Steps for safety PLC commissioning*)
		WAIT,
		CONNECT, (*Connection to the SafeDOMAIN*)
		LOAD_FILE, (*Load SafeCOMMISSIONING file*)
		PARA_SET, (*Set parameters to SafeCOMMISSIONING file*)
		NODE_AV, (*Set node availability to SafeCOMMISSIONING file*)
		SAVE_FILE, (*Save SafeCOMMISSIONING file*)
		TRANSFER, (*Transfer the SafeAPPLICATION and SafeCOMMISSIONING to the SafeDOMAIN*)
		READ_INFO, (*Read information from the SafeDOMAIN*)
		WAIT_ACK, (*Wait for acknowledgment*)
		COMPLETION, (*Completion Download*)
		DISCONNECT (*Disconnect from the SafeDOMAIN*)
		);
END_TYPE
```
